(* IEC 61131-3 sources: SmartHomeNew/snapshots/2026-04-28, 18 files *)

(* ---- E_Rule_Comparison.dut ---- *)
{attribute 'strict'}
TYPE E_Rule_Comparison :
(
    COMP_NONE := 0,
    COMP_EQ := 1,
    COMP_GT := 2,
    COMP_LT := 3,
    COMP_GE := 4,
    COMP_LE := 5,
    COMP_IN_RANGE := 6,
    COMP_TRUE := 7,
    COMP_FALSE := 8
) USINT;
END_TYPE

(* ---- E_SENSOR_TYPE.dut ---- *)
{attribute 'strict'}
TYPE E_SENSOR_TYPE :
(
  SENSOR_TYPE_NONE := 0,
  SENSOR_TYPE_DOOR_WINDOW := 5,
  SENSOR_TYPE_GLASS_BREAK := 6,
  SENSOR_TYPE_FLOOD := 7,
  SENSOR_TYPE_SMOKE := 8,
  SENSOR_TYPE_GAS_METHANE := 1,
  SENSOR_TYPE_GAS_CO := 2,
  SENSOR_TYPE_TEMP_FLOOR := 3,
  SENSOR_TYPE_TEMP_AIR := 4,
  SENSOR_TYPE_CO2 := 9
) USINT;
END_TYPE

(* ---- ST_Calibration_Family_Summary.dut ---- *)
{attribute 'pack_mode' := '1'}
TYPE ST_Calibration_Family_Summary :
STRUCT
    active : BOOL;
    status : INT; // 0=OK,1=IN_PROGRESS,2=WARNING,3=ERROR
    sensor_count : INT;
    verification_active_count : INT;
    failed_count : INT;
    max_deviation_percent : REAL;
    summary_text : STRING(160);
END_STRUCT
END_TYPE

(* ---- ST_Gas_Valve_Configuration.dut ---- *)
{attribute 'pack_mode' := '1'}
TYPE ST_Gas_Valve_Configuration :
STRUCT
    valve_id : BYTE := 0;
    valve_type : E_VALVE_TYPE := E_VALVE_TYPE.VALVE_NC;
    close_time_seconds : UDINT := 10;
    open_time_seconds : UDINT := 10;
    emergency_open_allowed : BOOL := FALSE;
END_STRUCT
END_TYPE

(* ---- GVL_HEATING_POLICY.gvl ---- *)
{attribute 'qualified_only'}
VAR_GLOBAL
    G_Zone_Empty_Duration_MS : ARRAY[1..GVL_CONSTANTS.C_MAX_ZONES] OF UDINT;
    G_Zone_Permanent_Use : ARRAY[1..GVL_CONSTANTS.C_MAX_ZONES] OF BOOL;
    G_Zone_Guest_Preheat_Request : ARRAY[1..GVL_CONSTANTS.C_MAX_ZONES] OF BOOL;
    G_Zone_Policy_Class : ARRAY[1..GVL_CONSTANTS.C_MAX_ZONES] OF INT;
    G_Zone_Target_Adjustment : ARRAY[1..GVL_CONSTANTS.C_MAX_ZONES] OF REAL;
    G_Zone_Priority_Bias : ARRAY[1..GVL_CONSTANTS.C_MAX_ZONES] OF REAL;
END_VAR

(* ---- GVL_HEATING_POLICY_CONFIG.gvl ---- *)
{attribute 'qualified_only'}
VAR_GLOBAL
    G_Guest_Preheat_Enabled : BOOL := TRUE;
    G_Guest_Preheat_Priority_Boost : INT := 2;
    G_Guest_Preheat_Max_Duration_MS : UDINT := 7200000; // 2 hours (future use)
END_VAR

(* ---- GVL_INTENT_USER.gvl ---- *)
VAR_GLOBAL
    I_Source_Valid : BOOL := FALSE;
    I_Last_Update_Cycle : UDINT := 0;
    I_Last_Update_MS : UDINT := 0;

    I_Arm_Request : BOOL := FALSE;
    I_Disarm_Request : BOOL := FALSE;

    I_PIN_Code : STRING(8);
    I_RFID_Tag : STRING(32);
    I_2FA_Code_In : STRING(8);

    I_Gate_Open_Request : BOOL := FALSE;
    I_Wicket_Open_Request : BOOL := FALSE;

    I_Lock_1_Open_Request : BOOL := FALSE;
    I_Lock_1_Close_Request : BOOL := FALSE;
    I_Lock_2_Open_Request : BOOL := FALSE;
    I_Lock_2_Close_Request : BOOL := FALSE;

    I_Dangerous_Action_Request : BOOL := FALSE;
    I_Dangerous_Action_Confirm : BOOL := FALSE;
    I_User_Access_Level : INT := 0;

    I_Water_Valve_Test_Open : BOOL := FALSE;
    I_Water_Valve_Test_Close : BOOL := FALSE;
    I_Water_Valve_Test_Confirm : BOOL := FALSE;

    I_Gas_Valve_Test_Open : BOOL := FALSE;
    I_Gas_Valve_Test_Close : BOOL := FALSE;
    I_Gas_Valve_Test_Confirm : BOOL := FALSE;

    I_Water_Selective_Recover : BOOL := FALSE;
    I_Gas_Selective_Recover : BOOL := FALSE;
    I_Scenario_Request : E_SCENARIO_TYPE := E_SCENARIO_TYPE.SCENARIO_NONE;
    I_Lighting_Override_32 : ARRAY[1..32] OF BYTE;
    I_Blinds_Override_32 : ARRAY[1..GVL_CONSTANTS.C_MAX_BLINDS] OF BYTE;
    I_Socket_Override_32 : ARRAY[1..GVL_CONSTANTS.C_MAX_SOCKETS] OF BOOL;
    I_Reset_Errors : BOOL := FALSE;

    I_Set_Temp_Req : BOOL := FALSE;
    I_Target_Zone : INT := 0;
    I_Target_Temperature : REAL := 0.0;
    I_Set_Vent_Req : BOOL := FALSE;
    I_Target_Vent_Speed : REAL := 0.0;
    I_Set_Config_Req : BOOL := FALSE;
    I_Time_Sync_Req : BOOL := FALSE;
    I_New_Time_MS : UDINT := 0;
END_VAR

(* ---- GVL_TEST_PANEL_DEBUG.gvl ---- *)
{attribute 'qualified_only'}
VAR_GLOBAL
    // === DEBUG VIEW ONLY ===
    G_Test_Description : STRING(200);
    G_Test_What_To_Change : STRING(200);
    G_Test_Expected_Text : STRING(200);
    G_Expected_Summary : STRING(200);
    G_Actual_Summary : STRING(200);
    G_Error_Text : STRING(200);
    G_System_State_Line : STRING(200);

    // Inputs snapshot
    G_Input_Guest_Preheat_Request : BOOL;
    G_Input_Guest_Preheat_Enabled : BOOL;
    G_Input_Guest_Preheat_Boost : INT;
    G_Input_Max_Thermal_Budget : REAL;
    G_Input_Block_Heating : BOOL;
    G_Input_Safety_Stop : BOOL;
END_VAR

(* ---- FB_Heating_System_Manager.st ---- *)
// ==============================================================================
// Блок управления системой отопления (Heating System Manager)
// Назначение:
// - Управление контурами теплого пола (открытие/закрытие клапанов).
// - Управление насосами коллекторов и смесительными узлами.
// - Управление каскадом котлов (ротация, расчет ресурса).
// - Защита от перегрева и замерзания.
// - Интеграция с Rule Engine.
// ==============================================================================
FUNCTION_BLOCK FB_Heating_System_Manager
VAR_INPUT
    VI_Preheat_Request : BOOL; // preheat scenario trigger
    L_Climate_Zone_ID : INT;

    VI_System_Mode : E_System_Operating_Mode; // System mode from State Manager

    VI_System_Time_MS : UDINT; // Системное время (мс)
    VI_Current_TOD : TOD; // Текущее время суток
    VI_IsActivePLC : BOOL; // Флаг: Данный ПЛК является ведущим
    VI_Outdoor_Temp : REAL; // Уличная температура воздуха (°C)
    VI_Config : ST_Heating_Config; // Конфигурация системы отопления
    VI_Tariff : ST_Tariff_Config; // Настройки тарифов
    VI_Current_Hour : UINT; // Текущий час (0-23)
    VI_Boiler_Stop : BOOL; // Команда на остановку котлов (от газовой/пожарной сигнализации); вход сохранён для совместимости, не используется как direct control
    VI_DHW_Heating_Demand : BOOL; // Запрос тепла от бойлера ГВС (приоритет)
    VI_DHW_Target_Temp : REAL; // Целевая температура бойлера ГВС
    VI_Current_Scenario : E_SCENARIO_TYPE; // Текущий сценарий
    VI_Emergency_Stop : BOOL; // Агрегированный аварийный стоп от подсистемы безопасности
    VI_Gas_Safety_Stop : BOOL; // Газовая авария / закрытие газового клапана
    VI_Boiler_Error_Status : ARRAY[1..GVL_CONSTANTS.C_MAX_BOILERS] OF BOOL; // Ошибки котлов / ошибка адаптера
    VI_Boiler_OT_Online : ARRAY[1..GVL_CONSTANTS.C_MAX_BOILERS] OF BOOL; // Признак доступности OpenTherm-канала
    VI_Boiler_Modulation : ARRAY[1..GVL_CONSTANTS.C_MAX_BOILERS] OF REAL; // Текущая модуляция котлов (%)
END_VAR
VAR_IN_OUT
    VI_Floor_Temps : ARRAY[1..GVL_CONSTANTS.C_MAX_HEATING_CIRCUITS] OF REAL; // Температуры стяжки пола по зонам
    VI_Room_Temps : ARRAY[1..16] OF REAL; // Температуры воздуха в помещениях
    VI_Manifold_Pressures : ARRAY[1..GVL_CONSTANTS.C_MAX_MANIFOLDS] OF REAL; // Давление в коллекторах (бар)
    VI_Manifold_Currents : ARRAY[1..GVL_CONSTANTS.C_MAX_MANIFOLDS] OF REAL; // Ток насосов коллекторов (мА)
    VI_Manifold_Temps_Supply : ARRAY[1..GVL_CONSTANTS.C_MAX_MANIFOLDS] OF REAL; // Температура подачи на коллекторах
    VI_Manifold_Temps_Return : ARRAY[1..GVL_CONSTANTS.C_MAX_MANIFOLDS] OF REAL; // Температура обратки на коллекторах
    VI_Boiler_Flame_Status : ARRAY[1..GVL_CONSTANTS.C_MAX_BOILERS] OF BOOL; // Статус наличия пламени в котлах
    VI_Zone_Configs : ARRAY[1..GVL_CONSTANTS.C_MAX_HEATING_CIRCUITS] OF ST_FloorHeating_Circuit_Config; // Конфигурации контуров
    VI_Rule_Actions : ARRAY[1..GVL_CONSTANTS.C_MAX_RULES] OF ST_Rule_Action; // Действия от Rule Engine
    VI_IO_Modules_Online : ARRAY[1..GVL_CONSTANTS.C_MAX_MODULES] OF BOOL; // Статусы модулей ввода-вывода
    VI_Scenario_Configs : ARRAY[1..GVL_CONSTANTS.C_MAX_SCENARIOS] OF ST_Scenario_Config; // Конфигурации сценариев
    VI_Manifold_End_Switches : ARRAY[1..GVL_CONSTANTS.C_MAX_MANIFOLDS] OF BOOL; // Концевики клапанов
    VI_Valve_Test_Config : ARRAY[1..GVL_CONSTANTS.C_MAX_MANIFOLDS] OF ST_Valve_Test_Config; // Конфигурация тестирования клапанов
END_VAR

VAR_OUTPUT
    VO_Manifold_Valves : ARRAY[1..GVL_CONSTANTS.C_MAX_MANIFOLDS] OF REAL; // Выход: Положение клапанов смесителей (0-100%)
    VO_Manifold_Pumps : ARRAY[1..GVL_CONSTANTS.C_MAX_MANIFOLDS] OF BOOL; // Выход: Управление насосами коллекторов
    VO_Zone_Valves : ARRAY[1..GVL_CONSTANTS.C_MAX_HEATING_CIRCUITS] OF BOOL; // Выход: Управление клапанами контуров (Зоны 1-16)
    VO_Boiler_OT_Enable : ARRAY[1..GVL_CONSTANTS.C_MAX_BOILERS] OF BOOL; // Физические команды в OpenTherm
    VO_Boiler_OT_Setpoint : ARRAY[1..GVL_CONSTANTS.C_MAX_BOILERS] OF REAL; // Физические уставки в OpenTherm
    VO_Backup_Circulation_Pump : BOOL; // Резервный циркуляционный насос в режиме антизамерзания при газовой аварии
    VO_Electric_Heater_Enable : BOOL; // Сухой контакт электрического нагревателя антизамерзания
    VO_Freeze_Risk_Status : BOOL; // Признак риска замерзания при защёлкнутой газовой аварии
    VO_Status : ARRAY[1..GVL_CONSTANTS.C_MAX_MANIFOLDS] OF ST_Manifold_Status; // Сводный статус коллекторных узлов для HMI
    VO_Boiler_Status : ARRAY[1..GVL_CONSTANTS.C_MAX_BOILERS] OF ST_Boiler_Status; // Сводный статус котлов для HMI
END_VAR

VAR

    L_PID_Valves : ARRAY[1..GVL_CONSTANTS.C_MAX_MANIFOLDS] OF FB_PID_Controller; // ПИД-регуляторы для поддержания температуры подачи
    L_PID_Timer : ARRAY[1..GVL_CONSTANTS.C_MAX_MANIFOLDS] OF FB_System_Timer; // Таймеры вызова ПИД-регуляторов
    L_Floor_Controllers : ARRAY[1..GVL_CONSTANTS.C_MAX_HEATING_CIRCUITS] OF FB_FloorHeating_Controller; // Контроллеры зон теплого пола
    L_Last_Boiler_Rotation : UDINT; // Время последней ротации ведущего котла
    L_Lead_Boiler : BYTE := 1; // Номер ведущего котла (1 или 2)
    L_i : INT; // Индекс для циклов
    L_Zone_Config : ST_FloorHeating_Circuit_Config;
    L_j : INT; // Вспомогательный индекс
    L_Target_Supply_Temp : REAL; // Рассчитанная целевая температура подачи
    L_Demand_Power : REAL; // Суммарный запрос мощности от всех коллекторов
    L_Any_Zone_Active : ARRAY[1..GVL_CONSTANTS.C_MAX_MANIFOLDS] OF BOOL; // Флаги наличия запроса тепла по коллекторам
    L_Current_Temp : REAL; // Текущая температура для ПИД
    L_Sensor_Error : BOOL; // Ошибка обоих датчиков

    // Плавный переход сценария
    L_Prev_Scenario : E_SCENARIO_TYPE;
    L_Scenario_Adjust : REAL;
    L_Target_Scenario_Adjust : REAL;
    L_Transition_Temp : FB_Scenario_Transition_Controller;

    // ТЗ 2.5: Защита от перегрева стяжки
    L_Overheat_Timer : ARRAY[1..GVL_CONSTANTS.C_MAX_HEATING_CIRCUITS] OF FB_System_Timer; // Таймеры задержки отключения при перегреве

    // ТЗ 2.6: Сервисная диагностика и паузы
    L_Pump_Run_Timer : ARRAY[1..GVL_CONSTANTS.C_MAX_MANIFOLDS] OF FB_System_Timer; // Таймер непрерывной работы насоса (до 72ч)
    L_Pump_Pause_Timer : ARRAY[1..GVL_CONSTANTS.C_MAX_MANIFOLDS] OF FB_System_Timer; // Таймер обязательной паузы насоса (1ч)
    L_Pump_In_Pause : ARRAY[1..GVL_CONSTANTS.C_MAX_MANIFOLDS] OF BOOL; // Флаг: Насос находится в режиме сервисной паузы

    // ТЗ 2.8: Учет ресурса оборудования
    L_Last_Scan_Time : UDINT; // Время предыдущего цикла для расчета наработки
    L_Scan_Time_Init : BOOL := FALSE;
    L_Lifespan_S : REAL := 50000.0 * 3600.0; // Расчетный ресурс котла (50,000 часов в секундах)
    L_Delta_MS : UDINT; // Разница времени
    L_Pump_Diag : ARRAY[1..GVL_CONSTANTS.C_MAX_MANIFOLDS] OF FB_Device_Predictive_Diag; // Диагностика насосов
    L_Boiler_Life : ARRAY[1..GVL_CONSTANTS.C_MAX_BOILERS] OF FB_Lifetime_Predictor; // Предиктор ресурса котлов

    fbFloorTempValidator : ARRAY[1..GVL_CONSTANTS.C_MAX_HEATING_CIRCUITS] OF FB_Analog_Validator;
    fbRoomTempValidator : ARRAY[1..16] OF FB_Analog_Validator;
    fbValveTestManager : FB_Valve_Test_Manager; // Менеджер тестирования клапанов
    fbBoilerCascade : FB_Boiler_Cascade_Manager; // Выделенный менеджер каскада котлов
    fbBoilerOpenTherm : FB_Boiler_OpenTherm_Interface; // Основной транспорт OpenTherm
    L_IO_Failsafe_Active : BOOL; // Флаг потери связи с модулями I/O
    L_Freeze_Mode_Active : BOOL; // Флаг антизамерзания по ТЗ
    L_Freeze_Target_Supply : REAL; // Уставка подачи в режиме антизамерзания
    L_Delta_T : REAL; // Разница температур подача/обратка
    L_Min_Supply_Temp : REAL; // Минимальная температура теплоносителя для антизамерзания
    L_Boiler_OT_Command_Valid : ARRAY[1..GVL_CONSTANTS.C_MAX_BOILERS] OF BOOL; // Команда ушла через OT
    L_Boiler_Request_Enable : ARRAY[1..GVL_CONSTANTS.C_MAX_BOILERS] OF BOOL; // Внутренний request на котлы от логики каскада
    L_Boiler_Request_Setpoint : ARRAY[1..GVL_CONSTANTS.C_MAX_BOILERS] OF REAL; // Внутренняя request-уставка котлов
    L_Policy_Normal : BOOL; // Policy: normal operation
    L_Policy_Safe_Stop : BOOL; // Policy: hard safe stop
    L_Policy_Degraded : BOOL; // Policy: limited conservative operation
    L_Policy_Freeze_Protection : BOOL; // Policy: freeze protection mode
    L_Any_Sensor_Error : BOOL;
    L_Any_Subsystem_Degraded : BOOL;
    L_Adaptive_Max_Delta : REAL;
    L_Adaptive_Delta : REAL;
    L_Adaptive_Zone_i : INT;
    L_Adaptive_Weighted_Sum : REAL;
    L_Adaptive_Weight_Total : REAL;
    L_Adaptive_Effective_Delta : REAL;
    L_Adaptive_Weight : REAL;
    L_Adaptive_Correction : REAL;
END_VAR

// ========================================
// Heating policy layer
// ========================================
L_Policy_Normal := (VI_System_Mode = E_System_Operating_Mode.MODE_NORMAL);
L_Policy_Safe_Stop := (VI_System_Mode = E_System_Operating_Mode.MODE_SAFE_STOP);
L_Policy_Degraded := (VI_System_Mode = E_System_Operating_Mode.MODE_DEGRADED);
L_Policy_Freeze_Protection := (VI_System_Mode = E_System_Operating_Mode.MODE_FREEZE_PROTECTION);

// ========================================
// Heating freeze policy activation
// ========================================
IF L_Policy_Freeze_Protection THEN
    L_Freeze_Mode_Active := TRUE;
END_IF;

// 0. Агрегация деградации для system mode
GVL_STATE.G_Heating_IO_Fault := FALSE;
GVL_STATE.G_Heating_Sensor_Fault := FALSE;
GVL_STATE.G_Heating_Subsystem_Degraded := FALSE;
L_Any_Sensor_Error := FALSE;
L_Any_Subsystem_Degraded := FALSE;

// 0. Аварийный стоп от подсистемы безопасности
VO_Backup_Circulation_Pump := FALSE;
VO_Electric_Heater_Enable := FALSE;
VO_Freeze_Risk_Status := FALSE;

IF VI_Gas_Safety_Stop THEN
    L_Freeze_Mode_Active := (VI_Outdoor_Temp < -5.0);
    FOR L_i := 1 TO GVL_CONSTANTS.C_MAX_HEATING_CIRCUITS DO
        IF VI_Floor_Temps[L_i] < 7.0 THEN
            L_Freeze_Mode_Active := TRUE;
        END_IF;
        VO_Zone_Valves[L_i] := FALSE;
    END_FOR;

    FOR L_i := 1 TO GVL_CONSTANTS.C_MAX_MANIFOLDS DO
        VO_Manifold_Pumps[L_i] := FALSE;
        VO_Manifold_Valves[L_i] := 0.0;
    END_FOR;

    FOR L_i := 1 TO GVL_CONSTANTS.C_MAX_BOILERS DO
        VO_Boiler_OT_Enable[L_i] := FALSE;
        VO_Boiler_OT_Setpoint[L_i] := 0.0;
        VO_Boiler_Status[L_i].Warning := FALSE;
        VO_Boiler_Status[L_i].Error := TRUE;
    END_FOR;

    IF L_Freeze_Mode_Active THEN
        VO_Backup_Circulation_Pump := TRUE;
        L_Freeze_Target_Supply := LIMIT(20.0, VI_Config.Freeze_Threshold + 2.0, 35.0);
        L_Min_Supply_Temp := 1000.0;
        FOR L_i := 1 TO GVL_CONSTANTS.C_MAX_MANIFOLDS DO
            IF VI_Manifold_Temps_Supply[L_i] < L_Min_Supply_Temp THEN
                L_Min_Supply_Temp := VI_Manifold_Temps_Supply[L_i];
            END_IF;
        END_FOR;
        IF L_Min_Supply_Temp > 900.0 THEN
            L_Min_Supply_Temp := 0.0;
        END_IF;

        IF L_Min_Supply_Temp < (L_Freeze_Target_Supply - 1.0) THEN
            VO_Electric_Heater_Enable := TRUE;
        ELSIF L_Min_Supply_Temp > (L_Freeze_Target_Supply + 1.0) THEN
            VO_Electric_Heater_Enable := FALSE;
        END_IF;

        // При защёлкнутой газовой аварии оператор должен видеть, что система живёт в деградированном anti-freeze режиме.
        VO_Freeze_Risk_Status := TRUE;
    END_IF;

    RETURN;
END_IF;

IF VI_Emergency_Stop OR L_Policy_Safe_Stop THEN
    FOR L_i := 1 TO GVL_CONSTANTS.C_MAX_HEATING_CIRCUITS DO
        VO_Zone_Valves[L_i] := FALSE;
    END_FOR;

    FOR L_i := 1 TO GVL_CONSTANTS.C_MAX_MANIFOLDS DO
        VO_Manifold_Pumps[L_i] := FALSE;
        VO_Manifold_Valves[L_i] := 0.0;
    END_FOR;

    FOR L_i := 1 TO GVL_CONSTANTS.C_MAX_BOILERS DO
        VO_Boiler_OT_Enable[L_i] := FALSE;
        VO_Boiler_OT_Setpoint[L_i] := 0.0;
        VO_Boiler_Status[L_i].Warning := FALSE;
        VO_Boiler_Status[L_i].Error := TRUE;
    END_FOR;

    RETURN;
END_IF;

// 1. Проверка связи с модулями ввода-вывода (ТЗ 2.0)
L_IO_Failsafe_Active := FALSE;
FOR L_i := 1 TO GVL_CONSTANTS.C_MAX_MODULES DO
    IF NOT VI_IO_Modules_Online[L_i] THEN
        L_IO_Failsafe_Active := TRUE;
        GVL_STATE.G_Heating_IO_Fault := TRUE;
GVL_STATE.G_Heating_Subsystem_Degraded := TRUE;
        EXIT;
    END_IF;
END_FOR;

IF L_IO_Failsafe_Active THEN
    // Fail-safe: закрываем зональные клапаны, чтобы не разгонять неконтролируемые контуры,
    // но при риске замерзания сохраняем минимальную циркуляцию и минимальную теплогенерацию.
    L_Freeze_Mode_Active := (VI_Outdoor_Temp < -5.0);

    FOR L_j := 1 TO GVL_CONSTANTS.C_MAX_HEATING_CIRCUITS DO
        IF VI_Floor_Temps[L_j] < 7.0 THEN
            L_Freeze_Mode_Active := TRUE;
        END_IF;
        VO_Zone_Valves[L_j] := FALSE;
    END_FOR;

    IF L_Freeze_Mode_Active THEN
        L_Freeze_Target_Supply := LIMIT(20.0, VI_Config.Freeze_Threshold + 2.0, 35.0);
    ELSE
        L_Freeze_Target_Supply := 0.0;
    END_IF;

    FOR L_j := 1 TO GVL_CONSTANTS.C_MAX_MANIFOLDS DO
        IF L_Freeze_Mode_Active THEN
            VO_Manifold_Pumps[L_j] := TRUE;
            VO_Manifold_Valves[L_j] := 35.0;
        ELSE
            VO_Manifold_Pumps[L_j] := FALSE;
            VO_Manifold_Valves[L_j] := 0.0;
        END_IF;
    END_FOR;

    // В аварийном I/O режиме напрямую формируем только legacy request-мirror.
    // Реальные физические команды всё равно будут интерпретированы transport-слоем выше по архитектуре.
    FOR L_j := 1 TO GVL_CONSTANTS.C_MAX_BOILERS DO
        VO_Boiler_OT_Enable[L_j] := FALSE;
        VO_Boiler_OT_Setpoint[L_j] := 0.0;
    END_FOR;

    IF L_Freeze_Mode_Active THEN
        // В fail-safe используем только ведущий аварийный вариант: котёл №1 на минимальной уставке.
        IF VI_Boiler_OT_Online[1] AND NOT VI_Boiler_Error_Status[1] THEN
            VO_Boiler_OT_Enable[1] := TRUE;
            VO_Boiler_OT_Setpoint[1] := L_Freeze_Target_Supply;
        END_IF;
    END_IF;

    RETURN;
END_IF;

// --- HEATING TARGET INJECTION ---
// Global arbitration target is applied after base policy calculation.
IF GVL_STATE.G_Target_Temperature > 0.0 THEN
    L_Target_Supply_Temp := GVL_STATE.G_Target_Temperature;
END_IF;

// --- MULTI-ZONE ADAPTIVE CORRECTION ---
// Final adaptive refinement layer.
L_Adaptive_Max_Delta := 0.0;
L_Adaptive_Weighted_Sum := 0.0;
L_Adaptive_Weight_Total := 0.0;
L_Adaptive_Effective_Delta := 0.0;
L_Adaptive_Correction := 0.0;

FOR L_Adaptive_Zone_i := 1 TO GVL_CONSTANTS.C_MAX_HEATING_CIRCUITS DO
    IF VI_Zone_Configs[L_Adaptive_Zone_i].zone >= 1 AND VI_Zone_Configs[L_Adaptive_Zone_i].zone <= 8 THEN
        CASE VI_Zone_Configs[L_Adaptive_Zone_i].control_type OF
            0:
                L_Adaptive_Delta :=
                    VI_Zone_Configs[L_Adaptive_Zone_i].design_temp -
                    VI_Floor_Temps[L_Adaptive_Zone_i];
                L_Adaptive_Weight := 0.6;
            1, 2:
                L_Adaptive_Delta :=
                    VI_Zone_Configs[L_Adaptive_Zone_i].design_temp -
                    VI_Room_Temps[VI_Zone_Configs[L_Adaptive_Zone_i].zone];
                L_Adaptive_Weight := 1.0;
            ELSE
                L_Adaptive_Delta :=
                    VI_Zone_Configs[L_Adaptive_Zone_i].design_temp -
                    VI_Room_Temps[VI_Zone_Configs[L_Adaptive_Zone_i].zone];
                L_Adaptive_Weight := 0.8;
        END_CASE;

        IF VI_Zone_Configs[L_Adaptive_Zone_i].zone >= 1 AND VI_Zone_Configs[L_Adaptive_Zone_i].zone <= 4 THEN
            L_Adaptive_Weight := L_Adaptive_Weight * 1.2;
        ELSIF VI_Zone_Configs[L_Adaptive_Zone_i].zone >= 9 THEN
            L_Adaptive_Weight := L_Adaptive_Weight * 0.7;
        END_IF;

        IF L_Adaptive_Weight > 2.0 THEN
            L_Adaptive_Weight := 2.0;
        ELSIF L_Adaptive_Weight < 0.2 THEN
            L_Adaptive_Weight := 0.2;
        END_IF;

        IF L_Adaptive_Delta > L_Adaptive_Max_Delta THEN
            L_Adaptive_Max_Delta := L_Adaptive_Delta;
        END_IF;

        L_Adaptive_Weighted_Sum := L_Adaptive_Weighted_Sum + (L_Adaptive_Delta * L_Adaptive_Weight);
        L_Adaptive_Weight_Total := L_Adaptive_Weight_Total + L_Adaptive_Weight;
    END_IF;
END_FOR;

IF L_Adaptive_Weight_Total > 0.0 THEN
    L_Adaptive_Effective_Delta := L_Adaptive_Weighted_Sum / L_Adaptive_Weight_Total;
END_IF;

IF L_Adaptive_Effective_Delta > 1.5 THEN
    L_Adaptive_Correction := 2.0;
ELSIF L_Adaptive_Effective_Delta > 0.7 THEN
    L_Adaptive_Correction := 1.0;
ELSIF L_Adaptive_Effective_Delta < -1.5 THEN
    L_Adaptive_Correction := -2.0;
ELSIF L_Adaptive_Effective_Delta < -0.7 THEN
    L_Adaptive_Correction := -1.0;
ELSE
    L_Adaptive_Correction := 0.0;
END_IF;

IF L_Adaptive_Max_Delta > 2.5 AND L_Adaptive_Correction < 2.0 THEN
    L_Adaptive_Correction := 2.0;
END_IF;

L_Target_Supply_Temp := L_Target_Supply_Temp + L_Adaptive_Correction;

IF L_Target_Supply_Temp < 20.0 THEN
    L_Target_Supply_Temp := 20.0;
ELSIF L_Target_Supply_Temp > 45.0 THEN
    L_Target_Supply_Temp := 45.0;
END_IF;

// 2. Индивидуальное управление зонами отопления (ТЗ 1.1, 2.5)
FOR L_i := 1 TO GVL_CONSTANTS.C_MAX_HEATING_CIRCUITS DO
    fbFloorTempValidator[L_i](
        VI_Value := VI_Floor_Temps[L_i],
        VI_Min_Valid := -40.0,
        VI_Max_Valid := 120.0,
        VI_Fallback_Mode := 0
    );

    L_Climate_Zone_ID := VI_Zone_Configs[L_i].zone;
    IF L_Climate_Zone_ID >= 1 AND L_Climate_Zone_ID <= 16 THEN
        fbRoomTempValidator[L_Climate_Zone_ID](
        VI_Value := VI_Room_Temps[L_Climate_Zone_ID],
        VI_Min_Valid := -40.0,
        VI_Max_Valid := 120.0,
        VI_Fallback_Mode := 0
        );
    END_IF;

    // Контроль перегрева стяжки (защита напольного покрытия)
    L_Overheat_Timer[L_i](IN := fbFloorTempValidator[L_i].VO_Value > VI_Config.Overheat_Threshold, PT := T#60s, VI_System_Time_MS := VI_System_Time_MS);

    // Выбор датчика температуры с автоматическим переключением при неисправности
    L_Current_Temp := 0.0;
    L_Sensor_Error := FALSE;

    IF VI_Zone_Configs[L_i].control_type = 1 OR VI_Zone_Configs[L_i].control_type = 2 THEN
        // Основной: по воздуху
        IF NOT fbRoomTempValidator[L_Climate_Zone_ID].VO_Error THEN
            L_Current_Temp := fbRoomTempValidator[L_Climate_Zone_ID].VO_Value;
        ELSIF NOT fbFloorTempValidator[L_i].VO_Error THEN
            L_Current_Temp := fbFloorTempValidator[L_i].VO_Value; // Резервный: по полу
        ELSE
            L_Sensor_Error := TRUE;
        END_IF;
    ELSE
        // Основной: по полу
        IF NOT fbFloorTempValidator[L_i].VO_Error THEN
            L_Current_Temp := fbFloorTempValidator[L_i].VO_Value;
        ELSIF NOT fbRoomTempValidator[L_Climate_Zone_ID].VO_Error THEN
            L_Current_Temp := fbRoomTempValidator[L_Climate_Zone_ID].VO_Value; // Резервный: по воздуху
        ELSE
            L_Sensor_Error := TRUE;
        END_IF;
    END_IF;

    IF L_Sensor_Error THEN
        L_Any_Sensor_Error := TRUE;
        VO_Zone_Valves[L_i] := FALSE; // Безопасное состояние при ошибке обоих датчиков
    ELSE
        // ПИД-регулирование и ШИМ для каждой зоны
        // Применяем плавную корректировку уставки от сценария
        L_Zone_Config := VI_Zone_Configs[L_i];
        L_Zone_Config.design_temp := L_Zone_Config.design_temp + L_Scenario_Adjust;
        L_Floor_Controllers[L_i](
            VI_Current_Temp := L_Current_Temp,
            VI_Config := L_Zone_Config,
            VI_Tariff := VI_Tariff,
            VI_Current_Hour := VI_Current_Hour,
            VI_IsActivePLC := VI_IsActivePLC,
            VI_System_Time_MS := VI_System_Time_MS,
            VO_Valve_Bool => VO_Zone_Valves[L_i]
        );
    END_IF;

    // Принудительное закрытие клапана при перегреве пола (ТЗ 2.5)
    IF L_Overheat_Timer[L_i].Q THEN
        VO_Zone_Valves[L_i] := FALSE;
    END_IF;

    // Обработка действий от Rule Engine (ТЗ 13.0)
    FOR L_j := 1 TO GVL_CONSTANTS.C_MAX_RULES DO
        IF VI_Rule_Actions[L_j].Active AND VI_Rule_Actions[L_j].Target_ID = L_i THEN
            IF VI_Rule_Actions[L_j].Action_Type = E_Rule_Action_Type.ACTION_SET_FLOOR_HEATING THEN
                VO_Zone_Valves[L_i] := (VI_Rule_Actions[L_j].Value > 0.5);
            END_IF;
        END_IF;
    END_FOR;
END_FOR;

GVL_STATE.G_Heating_Sensor_Fault := L_Any_Sensor_Error;

// 3. Определение потребности в работе коллекторных насосов
FOR L_i := 1 TO GVL_CONSTANTS.C_MAX_MANIFOLDS DO
    L_Any_Zone_Active[L_i] := FALSE;
END_FOR;

FOR L_i := 1 TO GVL_CONSTANTS.C_MAX_HEATING_CIRCUITS DO
    IF VO_Zone_Valves[L_i] THEN
        L_j := VI_Zone_Configs[L_i].manifold_id;
        IF L_j >= 1 AND L_j <= GVL_CONSTANTS.C_MAX_MANIFOLDS THEN
            L_Any_Zone_Active[L_j] := TRUE;
        END_IF;
    END_IF;
END_FOR;

// 4. Управление смесительными узлами коллекторов (ТЗ 2.6, 12.2)
FOR L_i := 1 TO GVL_CONSTANTS.C_MAX_MANIFOLDS DO
    // ПИД-регулирование трехходового клапана для поддержания стабильной температуры подачи
    // Вызываем ПИД регулятор каждую секунду
    L_PID_Timer[L_i](IN := TRUE, PT := T#1s, VI_System_Time_MS := VI_System_Time_MS);
    IF L_PID_Timer[L_i].Q THEN
        L_PID_Timer[L_i](IN := FALSE, PT := T#1s, VI_System_Time_MS := VI_System_Time_MS); // Сброс таймера
        L_PID_Timer[L_i](IN := TRUE, PT := T#1s, VI_System_Time_MS := VI_System_Time_MS); // Перезапуск

        L_PID_Valves[L_i](
            VI_SetPoint := L_Target_Supply_Temp,
            VI_ProcessValue := VI_Manifold_Temps_Supply[L_i],
            VI_Kp := 2.0, VI_Tn := 120.0, VI_Tv := 0.0,
            VI_Y_Min := 0.0, VI_Y_Max := 100.0, VI_Cycle_Time_S := 1.0,
            VO_Output => VO_Manifold_Valves[L_i]
        );
    END_IF;

    // ТЗ 2.6: Реализация обязательной паузы насоса (защита от закисания и перегрева при 72ч работе)
    L_Pump_Run_Timer[L_i](IN := VO_Manifold_Pumps[L_i] AND NOT L_Pump_In_Pause[L_i], PT := T#72h, VI_System_Time_MS := VI_System_Time_MS);
    IF L_Pump_Run_Timer[L_i].Q THEN L_Pump_In_Pause[L_i] := TRUE; END_IF;

    L_Pump_Pause_Timer[L_i](IN := L_Pump_In_Pause[L_i], PT := T#1h, VI_System_Time_MS := VI_System_Time_MS);
    IF L_Pump_Pause_Timer[L_i].Q THEN L_Pump_In_Pause[L_i] := FALSE; END_IF;

    // Включение насоса при наличии запроса от зон и отсутствии сервисной паузы
    // Приоритет ГВС: если есть запрос от ГВС, отключаем насосы отопления и закрываем клапаны
    IF VI_DHW_Heating_Demand THEN
        VO_Manifold_Pumps[L_i] := FALSE;
        VO_Manifold_Valves[L_i] := 0.0; // Принудительно закрываем смесительный клапан
    ELSE
        VO_Manifold_Pumps[L_i] := VI_IsActivePLC AND L_Any_Zone_Active[L_i] AND NOT L_Pump_In_Pause[L_i];
    END_IF;

    // Защита от замерзания системы (ТЗ 2.4)
        IF L_Freeze_Mode_Active THEN
            VO_Manifold_Pumps[L_i] := TRUE;
            IF VO_Manifold_Valves[L_i] < 35.0 THEN
                VO_Manifold_Valves[L_i] := 35.0;
            END_IF;
        END_IF;

        // Сбор диагностических данных для визуализации на HMI
    VO_Status[L_i].Pump_On := VO_Manifold_Pumps[L_i];
    VO_Status[L_i].Pump_Current := VI_Manifold_Currents[L_i];
    VO_Status[L_i].Pressure := VI_Manifold_Pressures[L_i];
    VO_Status[L_i].Temp_Supply := VI_Manifold_Temps_Supply[L_i];
    VO_Status[L_i].Temp_Return := VI_Manifold_Temps_Return[L_i];
    VO_Status[L_i].Valve_Pos := VO_Manifold_Valves[L_i];

    // Предиктивная диагностика насоса
    L_Pump_Diag[L_i](
        VI_Current_Value := VI_Manifold_Currents[L_i],
        VI_Nominal_Value := 0.55, // Номинальный ток насоса по ТЗ: середина диапазона 0.3..0.8 А
        VI_Is_Running := VO_Manifold_Pumps[L_i],
        VI_Reset_Stats := FALSE,
        VI_System_Time_MS := VI_System_Time_MS,
        VIO_Health_Data := VO_Status[L_i].Health
    );

    // Автоматический контроль рабочих параметров (ток / давление / ΔT)
        IF VO_Manifold_Pumps[L_i] THEN
            L_Delta_T := VI_Manifold_Temps_Supply[L_i] - VI_Manifold_Temps_Return[L_i];

            // Контроль тока насоса:
            // Приоритет ошибок:
            // 1. Насос/ток
            // 2. Давление
            // 3. ΔT
            VO_Status[L_i].Error := FALSE;
            VO_Status[L_i].Error_ID := 0;

            IF VI_Manifold_Currents[L_i] <= 0.01 THEN
                VO_Status[L_i].Error := TRUE;
                VO_Status[L_i].Error_ID := TO_WORD(GVL_CONFIG.ERR_PUMP_NO_CURRENT);
            ELSIF VI_Manifold_Currents[L_i] < 0.3 THEN
                VO_Status[L_i].Error := TRUE;
                VO_Status[L_i].Error_ID := TO_WORD(GVL_CONFIG.ERR_PUMP_UNDERCURRENT);
            ELSIF VI_Manifold_Currents[L_i] > 1.5 THEN
                VO_Status[L_i].Error := TRUE;
                VO_Status[L_i].Error_ID := TO_WORD(GVL_CONFIG.ERR_PUMP_OVERCURRENT);
            END_IF;

            // Проверка давления в системе (норма 1.5 - 2.5 бар)
            IF (NOT VO_Status[L_i].Error) AND (VI_Manifold_Pressures[L_i] < 1.5 OR VI_Manifold_Pressures[L_i] > 2.5) THEN
                VO_Status[L_i].Error := TRUE;
                VO_Status[L_i].Error_ID := TO_WORD(GVL_CONFIG.ERR_PRESSURE_OUT_OF_RANGE);
            END_IF;

            // Проверка эффективности теплообмена (ΔT 5..10°C норма)
            IF NOT VO_Status[L_i].Error THEN
                IF L_Delta_T < 5.0 THEN
                    VO_Status[L_i].Error := TRUE;
                    VO_Status[L_i].Error_ID := TO_WORD(GVL_CONFIG.ERR_DELTA_T_LOW);
                ELSIF L_Delta_T > 10.0 THEN
                    VO_Status[L_i].Error := TRUE;
                    VO_Status[L_i].Error_ID := TO_WORD(GVL_CONFIG.ERR_DELTA_T_HIGH);
                END_IF;
            END_IF;
        END_IF;

        // ТЗ 12.2: Еженедельное тестирование запорной арматуры (предотвращение закисания)
    // Выполняется менеджером fbValveTestManager
END_FOR;

fbValveTestManager(
    VI_System_Time_MS := VI_System_Time_MS,
    VI_IsActivePLC := VI_IsActivePLC,
    VI_Valve_Currents := VI_Manifold_Currents,
    VI_Valve_End_Switches := VI_Manifold_End_Switches,
    VI_Config := VI_Valve_Test_Config
);

IF fbValveTestManager.VO_Test_Active THEN
    L_i := fbValveTestManager.VO_Current_Valve;
    IF L_i >= 1 AND L_i <= GVL_CONSTANTS.C_MAX_MANIFOLDS THEN
        IF fbValveTestManager.VO_Valve_Cmd[L_i] THEN
            VO_Manifold_Valves[L_i] := 100.0;
        ELSE
            VO_Manifold_Valves[L_i] := 0.0;
        END_IF;
        VO_Manifold_Pumps[L_i] := FALSE; // Отключаем насос при тестировании клапана
    END_IF;
END_IF;

// 5. Управление каскадом котлов (ТЗ 2.8, OpenTherm-only, без legacy mirror)
L_Demand_Power := 0.0;
FOR L_i := 1 TO GVL_CONSTANTS.C_MAX_MANIFOLDS DO
    IF VO_Manifold_Pumps[L_i] THEN
        L_Demand_Power := L_Demand_Power + VO_Manifold_Valves[L_i];
    END_IF;
END_FOR;

// В режиме антизамерзания обеспечиваем минимальный запрос тепла
IF L_Freeze_Mode_Active AND L_Demand_Power < 20.0 THEN
    L_Demand_Power := 20.0;
END_IF;

IF L_Policy_Degraded THEN
    IF L_Demand_Power > 60.0 THEN
        L_Demand_Power := 60.0;
    END_IF;
END_IF;

fbBoilerCascade(
    VI_Enable := VI_IsActivePLC AND ((L_Demand_Power > GVL_CONSTANTS.C_BOILER_CASCADE_MIN_DEMAND) OR L_Freeze_Mode_Active),
    VI_System_Time_MS := VI_System_Time_MS,
    VI_Boiler_Stop := FALSE,
    VI_DHW_Heating_Demand := VI_DHW_Heating_Demand,
    VI_DHW_Target_Temp := VI_DHW_Target_Temp,
    VI_Target_Supply_Temp := L_Target_Supply_Temp,
    VI_Demand_Power := L_Demand_Power,
    VI_Boiler_Flame_Status := VI_Boiler_Flame_Status,
    VI_Boiler_Error_Status := VI_Boiler_Error_Status,
    VI_Boiler_OT_Online := VI_Boiler_OT_Online,
    VI_Boiler_Modulation := VI_Boiler_Modulation,
    VO_Boiler_Enable => L_Boiler_Request_Enable,
    VO_Boiler_Setpoint => L_Boiler_Request_Setpoint,
    VO_Lead_Boiler => L_Lead_Boiler
);

// ========================================
// OT availability enforcement (no fallback)
// ========================================
FOR L_i := 1 TO GVL_CONSTANTS.C_MAX_BOILERS DO
    IF NOT VI_Boiler_OT_Online[L_i] OR VI_Boiler_Error_Status[L_i] THEN
        L_Boiler_Request_Enable[L_i] := FALSE;
        L_Boiler_Request_Setpoint[L_i] := 0.0;
    END_IF;
END_FOR;

fbBoilerOpenTherm(
    VI_Enable := L_Boiler_Request_Enable,
    VI_Setpoint := L_Boiler_Request_Setpoint,
    VI_OT_Online := VI_Boiler_OT_Online,
    VI_OT_Error := VI_Boiler_Error_Status,
    VO_OT_Enable => VO_Boiler_OT_Enable,
    VO_OT_Setpoint => VO_Boiler_OT_Setpoint,
    VO_OT_Command_Valid => L_Boiler_OT_Command_Valid
);

// ========================================
// Boiler status normalization
// ========================================
FOR L_i := 1 TO GVL_CONSTANTS.C_MAX_BOILERS DO
    // Базовый сброс диагностических флагов котла
    VO_Boiler_Status[L_i].Active := L_Boiler_Request_Enable[L_i];
    VO_Boiler_Status[L_i].Warning := FALSE;
    VO_Boiler_Status[L_i].Error := FALSE;

    // Приоритет причин:
    // 1. Нет канала OpenTherm
    // 2. Котёл вернул ошибку
    // 3. Есть запрос, но нет пламени
    IF NOT VI_Boiler_OT_Online[L_i] THEN
        VO_Boiler_Status[L_i].Error := TRUE;
        VO_Boiler_Status[L_i].Error_ID := TO_WORD(GVL_CONFIG.ERR_BOILER_OFFLINE);
        L_Any_Subsystem_Degraded := TRUE;
    ELSIF VI_Boiler_Error_Status[L_i] THEN
        VO_Boiler_Status[L_i].Error := TRUE;
        VO_Boiler_Status[L_i].Error_ID := TO_WORD(GVL_CONFIG.ERR_BOILER_GENERAL_FAULT);
        L_Any_Subsystem_Degraded := TRUE;
    ELSIF L_Boiler_Request_Enable[L_i] AND NOT VI_Boiler_Flame_Status[L_i] THEN
        VO_Boiler_Status[L_i].Warning := TRUE;
        VO_Boiler_Status[L_i].Error_ID := TO_WORD(GVL_CONFIG.ERR_BOILER_NO_FLAME);
        L_Any_Subsystem_Degraded := TRUE;
    ELSE
        VO_Boiler_Status[L_i].Error_ID := 0;
    END_IF;
END_FOR;

// Расчет наработки и остаточного ресурса котлов (ТЗ 2.8)
IF NOT L_Scan_Time_Init THEN
    L_Last_Scan_Time := VI_System_Time_MS;
    L_Scan_Time_Init := TRUE;
END_IF;

L_Delta_MS := (SEL(VI_System_Time_MS >= L_Last_Scan_Time, VI_System_Time_MS - L_Last_Scan_Time, (4294967295 - L_Last_Scan_Time) + VI_System_Time_MS + 1));
IF L_Delta_MS > 1000 THEN
    L_Delta_MS := 1000; // Ограничение дельты для предотвращения скачков после перезагрузки
END_IF;

L_Last_Scan_Time := VI_System_Time_MS;

FOR L_i := 1 TO GVL_CONSTANTS.C_MAX_BOILERS DO
    VO_Boiler_Status[L_i].Work_Seconds := GVL_Retain.G_Boiler_Work_Seconds[L_i];

    IF VI_Boiler_Flame_Status[L_i] THEN
        GVL_Retain.G_Boiler_Accumulated_MS[L_i] := GVL_Retain.G_Boiler_Accumulated_MS[L_i] + L_Delta_MS;
        IF GVL_Retain.G_Boiler_Accumulated_MS[L_i] >= GVL_CONSTANTS.C_MS_IN_SECOND THEN
            GVL_Retain.G_Boiler_Work_Seconds[L_i] := GVL_Retain.G_Boiler_Work_Seconds[L_i] + (GVL_Retain.G_Boiler_Accumulated_MS[L_i] / 1000);
            GVL_Retain.G_Boiler_Accumulated_MS[L_i] := GVL_Retain.G_Boiler_Accumulated_MS[L_i] MOD 1000;

            // Защита от переполнения (сброс при достижении ~136 лет)
            IF GVL_Retain.G_Boiler_Work_Seconds[L_i] > 4000000000 THEN
                GVL_Retain.G_Boiler_Work_Seconds[L_i] := 0;
            END_IF;

            VO_Boiler_Status[L_i].Work_Seconds := GVL_Retain.G_Boiler_Work_Seconds[L_i];
        END_IF;
    END_IF;

    VO_Boiler_Status[L_i].Work_Hours := TO_REAL(VO_Boiler_Status[L_i].Work_Seconds) / 3600.0;

    L_Boiler_Life[L_i](
        VI_Runtime_Hours := TO_UDINT(VO_Boiler_Status[L_i].Work_Hours),
        VI_Start_Count := 0, // Не считаем пуски для котлов в этой версии
        VI_Nominal_Life := 50000 // 50,000 часов
    );
    VO_Boiler_Status[L_i].Resource_Percent := TO_REAL(L_Boiler_Life[L_i].VO_Remaining_Percent);
    VO_Boiler_Status[L_i].Running := VI_Boiler_Flame_Status[L_i];
END_FOR;
GVL_STATE.G_Heating_Subsystem_Degraded := L_Any_Subsystem_Degraded;

END_FUNCTION_BLOCK
// >>> BULK_SYNC_ANCHOR: FB_Heating_System_Manager <<<

(* ---- FB_Safety_Workflow_Manager.st ---- *)
FUNCTION_BLOCK FB_Safety_Workflow_Manager
VAR_INPUT
    VI_System_Time_MS : UDINT;
    VI_Water_Selective_Recover : BOOL;
    VI_Gas_Selective_Recover : BOOL;
    VI_Water_Valve_Test_Open : BOOL;
    VI_Water_Valve_Test_Close : BOOL;
    VI_Water_Valve_Test_Confirm : BOOL;
    VI_Gas_Valve_Test_Open : BOOL;
    VI_Gas_Valve_Test_Close : BOOL;
    VI_Gas_Valve_Test_Confirm : BOOL;
END_VAR
VAR_OUTPUT
    VO_Water_Selective_Recover_Edge : BOOL;
    VO_Gas_Selective_Recover_Edge : BOOL;
    VO_Water_Valve_Test_Open_Edge : BOOL;
    VO_Water_Valve_Test_Close_Edge : BOOL;
    VO_Water_Valve_Test_Confirm_Edge : BOOL;
    VO_Gas_Valve_Test_Open_Edge : BOOL;
    VO_Gas_Valve_Test_Close_Edge : BOOL;
    VO_Gas_Valve_Test_Confirm_Edge : BOOL;
    VO_Water_Test_Active : BOOL;
    VO_Gas_Test_Active : BOOL;
    VO_Water_Test_Timeout_Close_Required : BOOL;
    VO_Gas_Test_Timeout_Close_Required : BOOL;
END_VAR
VAR
    L_CMD_Water_Selective_Recover_Prev : BOOL;
    L_CMD_Gas_Selective_Recover_Prev : BOOL;
    L_CMD_Water_Valve_Test_Open_Prev : BOOL;
    L_CMD_Water_Valve_Test_Close_Prev : BOOL;
    L_CMD_Water_Valve_Test_Confirm_Prev : BOOL;
    L_CMD_Gas_Valve_Test_Open_Prev : BOOL;
    L_CMD_Gas_Valve_Test_Close_Prev : BOOL;
    L_CMD_Gas_Valve_Test_Confirm_Prev : BOOL;
    L_Water_Test_Active : BOOL;
    L_Water_Test_Deadline : UDINT;
    L_Gas_Test_Active : BOOL;
    L_Gas_Test_Deadline : UDINT;
END_VAR

VO_Water_Test_Timeout_Close_Required := FALSE;
VO_Gas_Test_Timeout_Close_Required := FALSE;

VO_Water_Selective_Recover_Edge := VI_Water_Selective_Recover AND NOT L_CMD_Water_Selective_Recover_Prev;
VO_Gas_Selective_Recover_Edge := VI_Gas_Selective_Recover AND NOT L_CMD_Gas_Selective_Recover_Prev;
VO_Water_Valve_Test_Open_Edge := VI_Water_Valve_Test_Open AND NOT L_CMD_Water_Valve_Test_Open_Prev;
VO_Water_Valve_Test_Close_Edge := VI_Water_Valve_Test_Close AND NOT L_CMD_Water_Valve_Test_Close_Prev;
VO_Water_Valve_Test_Confirm_Edge := VI_Water_Valve_Test_Confirm AND NOT L_CMD_Water_Valve_Test_Confirm_Prev;
VO_Gas_Valve_Test_Open_Edge := VI_Gas_Valve_Test_Open AND NOT L_CMD_Gas_Valve_Test_Open_Prev;
VO_Gas_Valve_Test_Close_Edge := VI_Gas_Valve_Test_Close AND NOT L_CMD_Gas_Valve_Test_Close_Prev;
VO_Gas_Valve_Test_Confirm_Edge := VI_Gas_Valve_Test_Confirm AND NOT L_CMD_Gas_Valve_Test_Confirm_Prev;

L_CMD_Water_Selective_Recover_Prev := VI_Water_Selective_Recover;
L_CMD_Gas_Selective_Recover_Prev := VI_Gas_Selective_Recover;
L_CMD_Water_Valve_Test_Open_Prev := VI_Water_Valve_Test_Open;
L_CMD_Water_Valve_Test_Close_Prev := VI_Water_Valve_Test_Close;
L_CMD_Water_Valve_Test_Confirm_Prev := VI_Water_Valve_Test_Confirm;
L_CMD_Gas_Valve_Test_Open_Prev := VI_Gas_Valve_Test_Open;
L_CMD_Gas_Valve_Test_Close_Prev := VI_Gas_Valve_Test_Close;
L_CMD_Gas_Valve_Test_Confirm_Prev := VI_Gas_Valve_Test_Confirm;

IF VO_Water_Valve_Test_Open_Edge THEN
    L_Water_Test_Active := TRUE;
    L_Water_Test_Deadline := VI_System_Time_MS + 60000;
END_IF;

IF L_Water_Test_Active THEN
    IF VI_System_Time_MS >= L_Water_Test_Deadline THEN
        L_Water_Test_Active := FALSE;
        VO_Water_Test_Timeout_Close_Required := TRUE;
    END_IF;
END_IF;

IF VO_Gas_Valve_Test_Open_Edge THEN
    L_Gas_Test_Active := TRUE;
    L_Gas_Test_Deadline := VI_System_Time_MS + 60000;
END_IF;

IF L_Gas_Test_Active THEN
    IF VI_System_Time_MS >= L_Gas_Test_Deadline THEN
        L_Gas_Test_Active := FALSE;
        VO_Gas_Test_Timeout_Close_Required := TRUE;
    END_IF;
END_IF;

VO_Water_Test_Active := L_Water_Test_Active;
VO_Gas_Test_Active := L_Gas_Test_Active;

(* ---- FB_State_Trace_Log.st ---- *)
FUNCTION_BLOCK FB_State_Trace_Log
VAR_INPUT
    VI_System_Time : UDINT;
    VI_Gas_Alarm : BOOL;
    VI_Leak_Alarm : BOOL;
    VI_Pumps : ARRAY[1..4] OF BOOL;
END_VAR
VAR_OUTPUT
    VO_Last_Change_Time : UDINT;
END_VAR
VAR
    L_Last_Gas : BOOL;
    L_Last_Leak : BOOL;
END_VAR

IF (VI_Gas_Alarm <> L_Last_Gas) OR (VI_Leak_Alarm <> L_Last_Leak) THEN
    VO_Last_Change_Time := VI_System_Time;
END_IF;

L_Last_Gas := VI_Gas_Alarm;
L_Last_Leak := VI_Leak_Alarm;

(* ---- FB_System_Timer_TOF.st ---- *)
// ==============================================================================
// Блок таймера задержки выключения (System Timer TOF)
// Назначение:
// - Замена стандартного TOF для обеспечения точной выдержки времени,
//   независимой от времени цикла ПЛК, с использованием единого системного времени.
// ==============================================================================
FUNCTION_BLOCK FB_System_Timer_TOF
VAR_INPUT
    IN : BOOL; // Вход запуска таймера
    PT : TIME; // Заданное время
    VI_System_Time_MS : UDINT; // Системное время (мс)
END_VAR
VAR_OUTPUT
    Q : BOOL; // Выход: таймер сработал
    ET : TIME; // Прошедшее время
END_VAR
VAR
    L_Start_Time : UDINT;
    L_Running : BOOL;
    L_Prev_IN : BOOL;
END_VAR

IF IN THEN
    Q := TRUE;
    ET := T#0s;
    L_Running := FALSE;
ELSE
    IF L_Prev_IN THEN
        L_Start_Time := VI_System_Time_MS;
        L_Running := TRUE;
        ET := T#0s;
    END_IF;

    IF L_Running THEN
        // Обработка переполнения UDINT (примерно 49 дней)
        ET := TO_TIME((SEL(VI_System_Time_MS >= L_Start_Time, VI_System_Time_MS - L_Start_Time, (4294967295 - L_Start_Time) + VI_System_Time_MS + 1)));

        IF ET >= PT THEN
            Q := FALSE;
            ET := PT;
            L_Running := FALSE;
        ELSE
            Q := TRUE;
        END_IF;
    END_IF;
END_IF;

L_Prev_IN := IN;

(* ---- PRG_IO_Read.st ---- *)
PROGRAM PRG_IO_Read
VAR
    L_i : INT;
    L_Debounce_Time : TIME := T#100MS;
    L_Manifold_Pressure_Raw : WORD;
    L_Manifold_Current_Raw : WORD;

    fbDebounce_Switches : ARRAY[1..8] OF FB_System_Timer;
    fbDebounce_Motion : ARRAY[1..8] OF FB_System_Timer;
    fbDebounce_Security_Open : ARRAY[1..GVL_CONSTANTS.C_MAX_SECURITY_SENSORS] OF FB_System_Timer;
    fbDebounce_Security_Glass : ARRAY[1..GVL_CONSTANTS.C_MAX_SECURITY_SENSORS] OF FB_System_Timer;
    fbDebounce_Flood : ARRAY[1..GVL_CONSTANTS.C_MAX_FLOOD_SENSORS] OF FB_System_Timer;
    fbDebounce_Smoke : ARRAY[1..GVL_CONSTANTS.C_MAX_SMOKE_SENSORS] OF FB_System_Timer;
    fbDebounce_Group_2F : FB_System_Timer;

    fbIO_Watchdog_1 : FB_IO_Module_Watchdog;
    fbIO_Watchdog_2 : FB_IO_Module_Watchdog;
    fbDiagEventManager : FB_Diagnostics_Event_Manager;
    L_IO_Error_Active : BOOL;

    // added
    fbCalib_Outdoor_Temp : FB_Sensor_Calibration_Processor;
    fbCalib_Supply_Temps : ARRAY[1..GVL_CONSTANTS.C_MAX_SUPPLY_TEMPS] OF FB_Sensor_Calibration_Processor;
    fbCalib_Room_Temps : ARRAY[1..GVL_CONSTANTS.C_MAX_ZONES] OF FB_Sensor_Calibration_Processor;
    fbCalib_Floor_Temps : ARRAY[1..GVL_CONSTANTS.C_MAX_ZONES] OF FB_Sensor_Calibration_Processor;
    fbCalib_Room_Hum : ARRAY[1..GVL_CONSTANTS.C_MAX_ZONES] OF FB_Sensor_Calibration_Processor;
    fbCalib_Room_CO2 : ARRAY[1..GVL_CONSTANTS.C_MAX_ZONES] OF FB_Sensor_Calibration_Processor;
    fbCalib_Manifold_T_Supply : ARRAY[1..GVL_CONSTANTS.C_MAX_MANIFOLDS] OF FB_Sensor_Calibration_Processor;
    fbCalib_Manifold_T_Return : ARRAY[1..GVL_CONSTANTS.C_MAX_MANIFOLDS] OF FB_Sensor_Calibration_Processor;
    fbCalib_Methane : ARRAY[1..GVL_CONSTANTS.C_MAX_METHANE_SENSORS] OF FB_Sensor_Calibration_Processor;
    fbCalib_CO : ARRAY[1..GVL_CONSTANTS.C_MAX_CO_SENSORS] OF FB_Sensor_Calibration_Processor;

    fbAnalog_Manifold_Pressure : ARRAY[1..GVL_CONSTANTS.C_MAX_MANIFOLDS] OF FB_Sensor_Analog_Processing;
    fbAnalog_Manifold_Current : ARRAY[1..GVL_CONSTANTS.C_MAX_MANIFOLDS] OF FB_Sensor_Analog_Processing;
END_VAR

// ===== ORIGINAL SNAPSHOT (FULL) =====
fbIO_Watchdog_1(VI_System_Time_MS := GVL_STATUS.G_System_Time_MS, VI_Module_ID := 1, VI_Heartbeat_Signal := GVL_IO.DI_Module_1_Heartbeat, VI_Timeout_MS := 2000);
fbIO_Watchdog_2(VI_System_Time_MS := GVL_STATUS.G_System_Time_MS, VI_Module_ID := 2, VI_Heartbeat_Signal := GVL_IO.DI_Module_2_Heartbeat, VI_Timeout_MS := 2000);

GVL_STATUS.G_IO_Modules_Online[1] := fbIO_Watchdog_1.VO_Module_Online;
GVL_STATUS.G_IO_Modules_Online[2] := fbIO_Watchdog_2.VO_Module_Online;

L_IO_Error_Active := fbIO_Watchdog_1.VO_Error_Active OR fbIO_Watchdog_2.VO_Error_Active;

// IO watchdog events
fbDiagEventManager(
    VI_Code := 16#E001,
    VI_Severity := 4,
    VI_Active := NOT fbIO_Watchdog_1.VO_Module_Online,
    VI_Timestamp := GVL_STATUS.G_System_Time_MS,
    VI_Source := 1,
    VIO_Events := GVL_STATUS.G_Diagnostics_Events,
    VIO_Count := GVL_STATUS.G_Diagnostics_Count
);

fbDiagEventManager(
    VI_Code := 16#E002,
    VI_Severity := 4,
    VI_Active := NOT fbIO_Watchdog_2.VO_Module_Online,
    VI_Timestamp := GVL_STATUS.G_System_Time_MS,
    VI_Source := 2,
    VIO_Events := GVL_STATUS.G_Diagnostics_Events,
    VIO_Count := GVL_STATUS.G_Diagnostics_Count
);

IF L_IO_Error_Active THEN
    GVL_COMMAND.G_Gas_Valve_Close := TRUE;
    GVL_COMMAND.G_Close_Valve_35 := TRUE;
    GVL_COMMAND.G_Close_Valve_36 := TRUE;
    FOR L_i := 1 TO GVL_CONSTANTS.C_MAX_MANIFOLDS DO GVL_STATE.G_Manifold_Pumps[L_i] := FALSE; END_FOR;
END_IF;

FOR L_i := 1 TO 8 DO
    fbDebounce_Switches[L_i](IN := GVL_IO.DI_Lighting_Switches[L_i], PT := L_Debounce_Time, VI_System_Time_MS := GVL_STATUS.G_System_Time_MS);
    GVL_STATE.G_Physical_Switches[L_i] := fbDebounce_Switches[L_i].Q;

    fbDebounce_Motion[L_i](IN := GVL_IO.DI_Motion_Sensors[L_i], PT := L_Debounce_Time, VI_System_Time_MS := GVL_STATUS.G_System_Time_MS);
    GVL_STATE.G_Motion_Sensors[L_i] := fbDebounce_Motion[L_i].Q;
END_FOR;

FOR L_i := 1 TO GVL_CONSTANTS.C_MAX_SOCKETS DO
    GVL_STATE.G_Socket_Switches[L_i] := FALSE;
END_FOR;

FOR L_i := 1 TO GVL_CONSTANTS.C_MAX_SECURITY_SENSORS DO
    fbDebounce_Security_Open[L_i](IN := GVL_IO.DI_Security_Open[L_i], PT := L_Debounce_Time, VI_System_Time_MS := GVL_STATUS.G_System_Time_MS);
    fbDebounce_Security_Glass[L_i](IN := GVL_IO.DI_Security_Glass[L_i], PT := L_Debounce_Time, VI_System_Time_MS := GVL_STATUS.G_System_Time_MS);
END_FOR;

fbDebounce_Group_2F(IN := GVL_IO.DI_Security_2F_Group, PT := L_Debounce_Time, VI_System_Time_MS := GVL_STATUS.G_System_Time_MS);

FOR L_i := 1 TO GVL_CONSTANTS.C_MAX_DOOR_SENSORS DO
    IF GVL_CONFIG.G_Door_Map[L_i] > 0 AND GVL_CONFIG.G_Door_Map[L_i] <= GVL_CONSTANTS.C_MAX_SECURITY_SENSORS THEN
        GVL_STATE.G_Door_Sensors[L_i] := fbDebounce_Security_Open[GVL_CONFIG.G_Door_Map[L_i]].Q;
    END_IF;
END_FOR;

FOR L_i := 1 TO 8 DO
    IF GVL_CONFIG.G_Window_Map[L_i] > 0 THEN
        IF GVL_CONFIG.G_Window_Map[L_i] <= GVL_CONSTANTS.C_MAX_SECURITY_SENSORS THEN
            GVL_STATE.G_Window_Sensors[L_i] := fbDebounce_Security_Open[GVL_CONFIG.G_Window_Map[L_i]].Q;
        ELSE
            GVL_STATE.G_Window_Sensors[L_i] := fbDebounce_Security_Glass[GVL_CONFIG.G_Window_Map[L_i] - GVL_CONSTANTS.C_MAX_SECURITY_SENSORS].Q;
        END_IF;
    END_IF;
END_FOR;
GVL_STATE.G_Window_Sensors[16] := fbDebounce_Group_2F.Q;

FOR L_i := 1 TO GVL_CONSTANTS.C_MAX_FLOOD_SENSORS DO
    fbDebounce_Flood[L_i](IN := GVL_IO.DI_Flood_Sensors[L_i], PT := L_Debounce_Time, VI_System_Time_MS := GVL_STATUS.G_System_Time_MS);
    GVL_STATE.G_Water_Sensors[L_i] := fbDebounce_Flood[L_i].Q;
END_FOR;

FOR L_i := 1 TO GVL_CONSTANTS.C_MAX_SMOKE_SENSORS DO
    fbDebounce_Smoke[L_i](IN := GVL_IO.DI_Smoke_Sensors[L_i], PT := L_Debounce_Time, VI_System_Time_MS := GVL_STATUS.G_System_Time_MS);
    GVL_STATE.G_Smoke_Sensors[L_i] := fbDebounce_Smoke[L_i].Q;
END_FOR;

// ===== ENHANCED LAYER =====
fbCalib_Outdoor_Temp(
    VI_Raw_Value := GVL_IO.AI_Temp_Outdoor.rValue,
    VI_Record := GVL_CONFIG.G_Calib_Outdoor_Temp
);
GVL_STATE.G_Outdoor_Temp := fbCalib_Outdoor_Temp.VO_Calibrated_Value;

FOR L_i := 1 TO GVL_CONSTANTS.C_MAX_SUPPLY_TEMPS DO
    IF GVL_IO.AI_Supply_Temps[L_i].wStatus = 0 THEN
        fbCalib_Supply_Temps[L_i](
            VI_Raw_Value := GVL_IO.AI_Supply_Temps[L_i].rValue,
            VI_Record := GVL_CONFIG.G_Calib_Supply_Temps[L_i]
        );
        GVL_STATE.G_Supply_Temps[L_i] := fbCalib_Supply_Temps[L_i].VO_Calibrated_Value;
    END_IF;
END_FOR;

FOR L_i := 1 TO 8 DO
    fbCalib_Room_Hum[L_i](
        VI_Raw_Value := GVL_IO.AI_Room_Hum[L_i],
        VI_Record := GVL_CONFIG.G_Calib_Humidity[L_i]
    );
    GVL_STATE.G_Room_Hum[L_i] := fbCalib_Room_Hum[L_i].VO_Calibrated_Value;

    fbCalib_Room_CO2[L_i](
        VI_Raw_Value := GVL_IO.AI_Room_CO2[L_i],
        VI_Record := GVL_CONFIG.G_Calib_CO2[L_i]
    );
    GVL_STATE.G_Room_CO2[L_i] := fbCalib_Room_CO2[L_i].VO_Calibrated_Value;
END_FOR;

FOR L_i := 1 TO 8 DO
    fbCalib_Room_Temps[L_i](
        VI_Raw_Value := GVL_IO.AI_Room_Temps[L_i],
        VI_Record := GVL_CONFIG.G_Calib_Room_Temps[L_i]
    );
    GVL_STATE.G_Room_Temps[L_i] := fbCalib_Room_Temps[L_i].VO_Calibrated_Value;

    fbCalib_Floor_Temps[L_i](
        VI_Raw_Value := GVL_IO.AI_Floor_Temps[L_i],
        VI_Record := GVL_CONFIG.G_Calib_Floor_Temps[L_i]
    );
    GVL_STATE.G_Floor_Temps[L_i] := fbCalib_Floor_Temps[L_i].VO_Calibrated_Value;
END_FOR;

GVL_STATUS.G_Diagnostics.Manifold_Pressure_Fault_Active := FALSE;
GVL_STATUS.G_Diagnostics.Manifold_Pressure_First_Fault_Index := 0;
GVL_STATUS.G_Diagnostics.Manifold_Current_Fault_Active := FALSE;
GVL_STATUS.G_Diagnostics.Manifold_Current_First_Fault_Index := 0;
GVL_STATUS.G_Diagnostics.Manifold_Pressure_Fault_Text := '';
GVL_STATUS.G_Diagnostics.Manifold_Current_Fault_Text := '';
GVL_STATUS.G_Diagnostics.Sensor_Fault := FALSE;
GVL_STATUS.G_Diagnostics.Subsystem_Degraded := FALSE;

FOR L_i := 1 TO GVL_CONSTANTS.C_MAX_MANIFOLDS DO
    IF GVL_IO.AI_Manifold_Pressures[L_i] < 0 THEN
        L_Manifold_Pressure_Raw := 0;
    ELSE
        L_Manifold_Pressure_Raw := INT_TO_WORD(GVL_IO.AI_Manifold_Pressures[L_i]);
    END_IF;

    IF GVL_IO.AI_Manifold_Currents[L_i] < 0 THEN
        L_Manifold_Current_Raw := 0;
    ELSE
        L_Manifold_Current_Raw := INT_TO_WORD(GVL_IO.AI_Manifold_Currents[L_i]);
    END_IF;

    fbAnalog_Manifold_Pressure[L_i](
        VI_Raw_Value := L_Manifold_Pressure_Raw,
        VI_Sensor_Type := 0,
        VI_Min_Scale := 0.0,
        VI_Max_Scale := 10.0,
        VI_Offset := 0.0,
        VI_Multiplier := 1.0,
        VI_Filter_Time_MS := GVL_CONSTANTS.C_MS_IN_SECOND,
        VI_System_Time_MS := GVL_STATUS.G_System_Time_MS,
        VI_Fallback_Mode := 0,
        VI_Default_Value := 0.0
    );
    GVL_STATE.G_Manifold_Pressures[L_i] := fbAnalog_Manifold_Pressure[L_i].VO_Value;
    GVL_STATUS.G_Diagnostics.Manifold_Pressure_Fault[L_i] := fbAnalog_Manifold_Pressure[L_i].VO_Error;
    GVL_STATUS.G_Diagnostics.Manifold_Pressure_Diag_Code[L_i] := fbAnalog_Manifold_Pressure[L_i].VO_Diag_Code;

    fbDiagEventManager(
        VI_Code := GVL_CONFIG.ERR_PRESSURE_OUT_OF_RANGE,
        VI_Severity := 3,
        VI_Active := fbAnalog_Manifold_Pressure[L_i].VO_Error,
        VI_Timestamp := GVL_STATUS.G_System_Time_MS,
        VI_Source := 100 + L_i,
        VIO_Events := GVL_STATUS.G_Diagnostics_Events,
        VIO_Count := GVL_STATUS.G_Diagnostics_Count
    );

    fbAnalog_Manifold_Current[L_i](
        VI_Raw_Value := L_Manifold_Current_Raw,
        VI_Sensor_Type := 0,
        VI_Min_Scale := 0.0,
        VI_Max_Scale := 16.0,
        VI_Offset := 0.0,
        VI_Multiplier := 1.0,
        VI_Filter_Time_MS := GVL_CONSTANTS.C_MS_IN_SECOND,
        VI_System_Time_MS := GVL_STATUS.G_System_Time_MS,
        VI_Fallback_Mode := 0,
        VI_Default_Value := 0.0
    );
    GVL_STATE.G_Manifold_Currents[L_i] := fbAnalog_Manifold_Current[L_i].VO_Value;
    GVL_STATUS.G_Diagnostics.Manifold_Current_Fault[L_i] := fbAnalog_Manifold_Current[L_i].VO_Error;
    GVL_STATUS.G_Diagnostics.Manifold_Current_Diag_Code[L_i] := fbAnalog_Manifold_Current[L_i].VO_Diag_Code;

    fbDiagEventManager(
        VI_Code := GVL_CONFIG.ERR_PUMP_UNDERCURRENT,
        VI_Severity := 3,
        VI_Active := fbAnalog_Manifold_Current[L_i].VO_Error,
        VI_Timestamp := GVL_STATUS.G_System_Time_MS,
        VI_Source := 200 + L_i,
        VIO_Events := GVL_STATUS.G_Diagnostics_Events,
        VIO_Count := GVL_STATUS.G_Diagnostics_Count
    );

    IF GVL_IO.AI_Manifold_Temps_Supply[L_i].wStatus = 0 THEN
        fbCalib_Manifold_T_Supply[L_i](
            VI_Raw_Value := GVL_IO.AI_Manifold_Temps_Supply[L_i].rValue,
            VI_Record := GVL_CONFIG.G_Calib_Manifold_T_Supply[L_i]
        );
        GVL_STATE.G_Manifold_T_Supply[L_i] := fbCalib_Manifold_T_Supply[L_i].VO_Calibrated_Value;
    END_IF;

    fbCalib_Manifold_T_Return[L_i](
        VI_Raw_Value := INT_TO_REAL(GVL_IO.AI_Manifold_Temps_Return[L_i]) / 10.0,
        VI_Record := GVL_CONFIG.G_Calib_Manifold_T_Return[L_i]
    );
    GVL_STATE.G_Manifold_T_Return[L_i] := fbCalib_Manifold_T_Return[L_i].VO_Calibrated_Value;
    GVL_STATE.G_Manifold_End_Switches[L_i] := GVL_IO.DI_Manifold_End_Switches[L_i];

    IF GVL_STATUS.G_Diagnostics.Manifold_Pressure_Fault[L_i] OR GVL_STATUS.G_Diagnostics.Manifold_Current_Fault[L_i] THEN
        GVL_STATUS.G_Diagnostics.Sensor_Fault := TRUE;
        GVL_STATUS.G_Diagnostics.Subsystem_Degraded := TRUE;
    END_IF;

    IF GVL_STATUS.G_Diagnostics.Manifold_Pressure_Fault[L_i] AND GVL_STATUS.G_Diagnostics.Manifold_Current_Fault[L_i] THEN
        GVL_STATUS.G_Diagnostics.Manifold_Pressure_Fault_Text := 'Correlated pressure/current fault detected';
        GVL_STATUS.G_Diagnostics.Manifold_Current_Fault_Text := 'Correlated pressure/current fault detected';
    ELSIF GVL_STATUS.G_Diagnostics.Manifold_Pressure_Fault[L_i] AND (GVL_STATUS.G_Diagnostics.Manifold_Pressure_Fault_Text = '') THEN
        GVL_STATUS.G_Diagnostics.Manifold_Pressure_Fault_Text := 'Pressure sensor fault detected';
    ELSIF GVL_STATUS.G_Diagnostics.Manifold_Current_Fault[L_i] AND (GVL_STATUS.G_Diagnostics.Manifold_Current_Fault_Text = '') THEN
        GVL_STATUS.G_Diagnostics.Manifold_Current_Fault_Text := 'Current sensor fault detected';
    END_IF;
END_FOR;

FOR L_i := 1 TO GVL_CONSTANTS.C_MAX_METHANE_SENSORS DO
    IF GVL_IO.AI_Methane_LEL[L_i].wStatus = 0 THEN
        fbCalib_Methane[L_i](
            VI_Raw_Value := GVL_IO.AI_Methane_LEL[L_i].rValue,
            VI_Record := GVL_CONFIG.G_Calib_Methane[L_i]
        );
        GVL_STATE.G_Methane_Sensors[L_i] := fbCalib_Methane[L_i].VO_Calibrated_Value;
    END_IF;

    fbDiagEventManager(
        VI_Code := 16#E003,
        VI_Severity := 3,
        VI_Active := GVL_IO.AI_Methane_LEL[L_i].wStatus <> 0,
        VI_Timestamp := GVL_STATUS.G_System_Time_MS,
        VI_Source := 300 + L_i,
        VIO_Events := GVL_STATUS.G_Diagnostics_Events,
        VIO_Count := GVL_STATUS.G_Diagnostics_Count
    );
END_FOR;

FOR L_i := 1 TO GVL_CONSTANTS.C_MAX_CO_SENSORS DO
    fbCalib_CO[L_i](
        VI_Raw_Value := GVL_IO.AI_CO_PPM[L_i],
        VI_Record := GVL_CONFIG.G_Calib_CO[L_i]
    );
    GVL_STATE.G_CO_Sensors[L_i] := fbCalib_CO[L_i].VO_Calibrated_Value;
END_FOR;

GVL_STATE.G_Boiler_Flame := GVL_IO.AI_Boiler_Flame_Status;
GVL_STATE.G_Boiler_Error := GVL_IO.DI_Boiler_Error;
FOR L_i := 1 TO GVL_CONSTANTS.C_MAX_BOILERS DO
    GVL_STATE.G_Boiler_OT_Online[L_i] := FALSE;
END_FOR;

GVL_STATE.G_DHW_Temp := GVL_IO.AI_DHW_Temp;
GVL_STATE.G_DHW_Pressure := GVL_IO.AI_DHW_Pressure;

GVL_STATE.G_Water_Zone_Open_FB := GVL_IO.DI_Water_Zone_Open_FB;
GVL_STATE.G_Water_Zone_Close_FB := GVL_IO.DI_Water_Zone_Close_FB;

// >>> BULK_SYNC_ANCHOR: PRG_IO_Read <<<

(* ---- PRG_IO_Write.st ---- *)
PROGRAM PRG_IO_Write
VAR
    L_i : INT;
END_VAR

// 2. ЗАПИСЬ ВЫХОДОВ (GVL_STATE -> GVL_IO)

// 2.1. Отопление (Термоэлектрические приводы)
FOR L_i := 1 TO 8 DO
    GVL_IO.DO_Zone_Valves[L_i] := GVL_STATE.G_Zone_Valves[L_i];
END_FOR;

// 2.2. Коллекторы (Насосы и смесительные клапаны)
FOR L_i := 1 TO GVL_CONSTANTS.C_MAX_MANIFOLDS DO
    GVL_IO.DO_Manifold_Pumps[L_i] := GVL_STATE.G_Manifold_Pumps[L_i];
    GVL_IO.AO_Manifold_Valves[L_i] := REAL_TO_UINT(GVL_STATE.G_Manifold_Valves[L_i] * 1000.0);
END_FOR;

// 2.4. Вентиляция
FOR L_i := 1 TO GVL_CONSTANTS.C_MAX_SUPPLY_FANS DO
    GVL_IO.AO_Supply_Fans[L_i] := REAL_TO_UINT(GVL_STATE.G_Supply_Fans[L_i] * 100.0);
END_FOR;
FOR L_i := 1 TO GVL_CONSTANTS.C_MAX_EXHAUST_FANS DO
    GVL_IO.AO_Exhaust_Fans[L_i] := REAL_TO_UINT(GVL_STATE.G_Exhaust_Fans[L_i] * 100.0);
END_FOR;

// 2.5. ГВС
GVL_IO.DO_DHW_Heating_Pump := GVL_STATE.G_DHW_Heating_Pump;
GVL_IO.DO_DHW_Circ_Pump := GVL_STATE.G_DHW_Circ_Pump;
IF GVL_STATUS.G_Is_Active_PLC THEN
    GVL_IO.DO_Backup_Circulation_Pump := GVL_STATE.G_Backup_Circulation_Pump;
    GVL_IO.DO_Electric_Heater_Enable := GVL_STATE.G_Electric_Heater_Enable;
ELSE
    GVL_IO.DO_Backup_Circulation_Pump := FALSE;
    GVL_IO.DO_Electric_Heater_Enable := FALSE;
END_IF;

// 2.6. Освещение и шторы
FOR L_i := 1 TO 8 DO
    GVL_IO.AO_Lighting_Levels[L_i] := BYTE_TO_UINT(GVL_STATE.G_Lighting_Levels[L_i]) * 10;
END_FOR;
FOR L_i := 1 TO GVL_CONSTANTS.C_MAX_BLINDS DO
    GVL_IO.AO_Blinds_Positions[L_i] := BYTE_TO_UINT(GVL_STATE.G_Blinds_Positions[L_i]) * 10;
END_FOR;

// 2.7. Аварийные выходы (Сирены и клапаны)
GVL_IO.DO_Gas_Siren := (GVL_ALARM.G_Gas_Fire_Siren AND GVL_ALARM.G_Gas_Alarm_Active);
GVL_IO.DO_Fire_Siren := (GVL_ALARM.G_Gas_Fire_Siren AND GVL_ALARM.G_Fire_Alarm_Active);
GVL_IO.DO_Security_Siren := GVL_ALARM.G_Security_Siren;

// === STAGE H2: USE SHADOW COMMANDS ===
GVL_IO.DO_Water_Valve_35_Close := GVL_COMMAND_SHADOW.G_Close_Valve_35;
GVL_IO.DO_Water_Valve_36_Close := GVL_COMMAND_SHADOW.G_Close_Valve_36;
GVL_IO.DO_Gas_Valve_Close := GVL_COMMAND_SHADOW.G_Gas_Valve_Close;

// Access control (shadow)
GVL_IO.DO_Lock_1_Open := GVL_COMMAND_SHADOW.G_Lock_1_Open;
GVL_IO.DO_Lock_1_Close := GVL_COMMAND_SHADOW.G_Lock_1_Close;
GVL_IO.DO_Lock_2_Open := GVL_COMMAND_SHADOW.G_Lock_2_Open;
GVL_IO.DO_Lock_2_Close := GVL_COMMAND_SHADOW.G_Lock_2_Close;

// Gate/Wicket — now via shadow
GVL_IO.DO_Gate_Open := GVL_COMMAND_SHADOW.G_Gate_Open;
GVL_IO.DO_Wicket_Open := GVL_COMMAND_SHADOW.G_Wicket_Open;

// 2.9. Розетки
GVL_IO.DO_Sockets := GVL_STATE.G_Socket_States;

// Selective zonal water recovery outputs
FOR L_i := 1 TO 32 DO
    GVL_IO.DO_Water_Zone_Enable[L_i] := GVL_STATE.G_Water_Zone_Enable[L_i];
END_FOR;

// >>> BULK_SYNC_ANCHOR: PRG_IO_Write <<<

(* ---- PRG_Lighting.st ---- *)
PROGRAM PRG_Lighting
VAR
    L_i : INT;
    fbLightingManager : FB_Lighting_Blinds_Manager;
    fbSocketManager : FB_Socket_Manager;
    L_Manual_Light_Override_32 : ARRAY[1..32] OF BYTE;
    L_Manual_Blinds_Override_32 : ARRAY[1..32] OF BYTE;
    L_Manual_Socket_Override_32 : ARRAY[1..32] OF BOOL;
    L_Sim_Lights_32 : ARRAY[1..32] OF BOOL;
    L_Physical_Switches_32 : ARRAY[1..32] OF BOOL;
    L_Motion_Sensors_32 : ARRAY[1..32] OF BOOL;

    // ADAPTER ARRAYS (match FB expected sizes)
    L_Blinds_Override : ARRAY[1..GVL_CONSTANTS.C_MAX_BLINDS] OF BYTE;
    L_Socket_Override : ARRAY[1..GVL_CONSTANTS.C_MAX_SOCKETS] OF BOOL;
END_VAR

FOR L_i := 1 TO 32 DO
    IF L_i <= 16 THEN
        IF GVL_INTENT_SYSTEM.I_Lighting_Overrides_Block OR GVL_SYSTEM_COORDINATION.G_Block_Lighting_Override THEN
            L_Manual_Light_Override_32[L_i] := 0;
        ELSE
            L_Manual_Light_Override_32[L_i] := GVL_INTENT_USER.I_Lighting_Override_32[L_i];
        END_IF;
        L_Sim_Lights_32[L_i] := GVL_STATE.G_Sim_Lights[L_i];
        L_Physical_Switches_32[L_i] := GVL_STATE.G_Physical_Switches[L_i];
        L_Motion_Sensors_32[L_i] := GVL_STATE.G_Motion_Sensors[L_i];
    ELSE
        L_Manual_Light_Override_32[L_i] := 0;
        L_Sim_Lights_32[L_i] := FALSE;
        L_Physical_Switches_32[L_i] := FALSE;
        L_Motion_Sensors_32[L_i] := FALSE;
    END_IF;

    IF GVL_INTENT_SYSTEM.I_Blinds_Overrides_Block THEN
        L_Manual_Blinds_Override_32[L_i] := 0;
    ELSE
        L_Manual_Blinds_Override_32[L_i] := GVL_INTENT_USER.I_Blinds_Override_32[L_i];
    END_IF;

    IF GVL_INTENT_SYSTEM.I_Socket_Overrides_Block OR GVL_SYSTEM_COORDINATION.G_Block_Sockets_Override THEN
        L_Manual_Socket_Override_32[L_i] := FALSE;
    ELSE
        L_Manual_Socket_Override_32[L_i] := GVL_INTENT_USER.I_Socket_Override_32[L_i];
    END_IF;
END_FOR;

// ADAPTER: copy to FB-sized arrays
FOR L_i := 1 TO GVL_CONSTANTS.C_MAX_BLINDS DO
    L_Blinds_Override[L_i] := L_Manual_Blinds_Override_32[L_i];
END_FOR;

FOR L_i := 1 TO GVL_CONSTANTS.C_MAX_SOCKETS DO
    L_Socket_Override[L_i] := L_Manual_Socket_Override_32[L_i];
END_FOR;

// 10. Управление освещением и шторами
fbLightingManager(
    VI_System_Time_MS := GVL_STATUS.G_System_Time_MS,
    VI_IsActivePLC := GVL_STATUS.G_Is_Active_PLC,
    VI_Current_Scenario := GVL_STATUS.G_Current_Scenario,
    VI_Away_Level := 1,
    VI_Simulation_Active := GVL_STATUS.G_Sim_Active,
    VI_Manual_Light_Override := L_Manual_Light_Override_32,
    VI_Manual_Blinds_Override := L_Blinds_Override,
    VI_Simulation_Lights := L_Sim_Lights_32,
    VI_Physical_Switches := L_Physical_Switches_32,
    VI_Motion_Sensors := L_Motion_Sensors_32,
    VI_Is_Night := GVL_STATUS.G_Is_Night,
    VI_Rule_Actions := GVL_STATE.G_Rule_Actions,
    VI_IO_Modules_Online := GVL_STATUS.G_IO_Modules_Online,
    VI_Wet_Zone_Map := GVL_CONFIG.G_Wet_Zone_Map,
    VI_Scenario_Configs := GVL_CONFIG.G_HMI_Scenario_Configs,
    VO_Lighting_Levels => GVL_STATE.G_Lighting_Levels,
    VO_Blinds_Positions => GVL_STATE.G_Blinds_Positions
);

// 11.5 Управление розетками
fbSocketManager(
    VI_System_Time_MS := GVL_STATUS.G_System_Time_MS,
    VI_IsActivePLC := GVL_STATUS.G_Is_Active_PLC,
    VI_Scenario := GVL_STATUS.G_Current_Scenario,
    VI_Manual_Override := L_Socket_Override,
    VI_Physical_Switches := GVL_STATE.G_Socket_Switches,
    VI_Rule_Actions := GVL_STATE.G_Rule_Actions,
    VI_Fire_Alarm := GVL_ALARM.G_Fire_Alarm_Active,
    VI_Flood_Alarm := GVL_ALARM.G_Flood_Alarm_Active,
    VI_Security_Armed := GVL_ALARM.G_Security_Armed,
    VI_IO_Modules_Online := GVL_STATUS.G_IO_Modules_Online,
    VO_Socket_States => GVL_STATE.G_Socket_States
);

// Evacuation lighting override
IF GVL_STATE.G_Evacuation_Lighting_Active THEN
    FOR L_i := 1 TO 8 DO
        IF (L_i MOD 2) = 0 THEN
            GVL_STATE.G_Lighting_Levels[L_i] := 100;
        ELSE
            GVL_STATE.G_Lighting_Levels[L_i] := 0;
        END_IF;
    END_FOR;
END_IF;

// Directional evacuation override
IF GVL_STATE.G_Evacuation_Lighting_Active THEN
    FOR L_i := 1 TO GVL_CONFIG.C_MAX_LIGHT_ZONES DO
        CASE GVL_STATE.G_Evac_Guidance[L_i] OF
            -1:
                GVL_STATE.G_Lighting_Levels[L_i] := 0;
            1:
                GVL_STATE.G_Lighting_Levels[L_i] := 100;
        ELSE
            GVL_STATE.G_Lighting_Levels[L_i] := SEL((L_i MOD 2) = 0, 0, 100);
        END_CASE;
    END_FOR;
END_IF;
// >>> BULK_SYNC_ANCHOR: PRG_Lighting <<<

(* ---- PRG_Presence_Manager.st ---- *)
PROGRAM PRG_Presence_Manager
VAR
    fbPresence : FB_Presence_Manager;
    L_i : INT;
END_VAR

fbPresence(
    VI_Motion_Sensors := GVL_STATE.G_Motion_Sensors,
    VI_System_Time_MS := GVL_STATUS.G_System_Time_MS
);

GVL_PRESENCE.G_Any_Motion := fbPresence.VO_Any_Motion;
GVL_PRESENCE.G_Occupied := fbPresence.VO_Occupied;
GVL_PRESENCE.G_Auto_Away_Request := fbPresence.VO_Auto_Away;
GVL_PRESENCE.G_Last_Motion_TS := fbPresence.VO_Last_Motion_TS;

FOR L_i := 1 TO GVL_CONSTANTS.C_MAX_ZONES DO
    IF GVL_STATE.G_Motion_Sensors[L_i] THEN
        GVL_PRESENCE.G_Zone_Occupied[L_i] := TRUE;
        GVL_PRESENCE.G_Zone_Last_Motion_TS[L_i] := GVL_STATUS.G_System_Time_MS;
    END_IF;

    IF (GVL_STATUS.G_System_Time_MS - GVL_PRESENCE.G_Zone_Last_Motion_TS[L_i]) > 900000 THEN
        GVL_PRESENCE.G_Zone_Occupied[L_i] := FALSE;
    END_IF;
END_FOR;

(* ---- PRG_System_Test_Harness.st ---- *)
PROGRAM PRG_System_Test_Harness
VAR
    L_i : INT;
    L_j : INT;
    L_Used : REAL;
    L_HP_Used : REAL;
    L_HP_Manifold_Adjusted : ARRAY[1..GVL_CONSTANTS.C_MAX_MANIFOLDS] OF INT;
    fbDecisionTest : FB_Heating_Decision_Context;
    fbDecisionHP : FB_Heating_Decision_Context;
    fbTestResult : FB_Test_Result_Handler;
    fbTrace : FB_Trace_Logger;
END_VAR

IF NOT GVL_TEST.G_Test_Enable THEN
    RETURN;
END_IF;

GVL_TEST.G_Test_Total_Checks := 0;
GVL_TEST.G_Test_Failed_Checks := 0;
GVL_TEST.G_Test_Passed := TRUE;
GVL_TEST.G_Test_Last_Failure_Index := 0;
GVL_TEST.G_Test_Last_Failure_Code := 0;

// Reset transient failure flags for this scan
GVL_TEST.G_Diagnostics_Duplicate_Event_Found := FALSE;
GVL_TEST.G_Diagnostics_Count_Out_Of_Range := FALSE;
GVL_TEST.G_Heating_Allocation_Budget_Exceeded := FALSE;
GVL_TEST.G_Heating_Allocation_Enabled_Not_Allowed := FALSE;
GVL_TEST.G_Safety_Latched_Without_Intent := FALSE;
GVL_TEST.G_HP_Adjusted_Priority_Lower_Bound_Violation := FALSE;
GVL_TEST.G_HP_Adjusted_Allocation_Budget_Exceeded := FALSE;
GVL_TEST.G_HP_Adjusted_Allocation_Enabled_Not_Allowed := FALSE;
GVL_TEST.G_HP_Guest_Preheat_Config_Out_Of_Range := FALSE;

// =========================
// TEST 1: Diagnostics count bounds
// =========================
GVL_TEST.G_Test_Total_Checks := GVL_TEST.G_Test_Total_Checks + 1;
IF (GVL_STATUS.G_Diagnostics_Count < 0) OR (GVL_STATUS.G_Diagnostics_Count > 50) THEN
    GVL_TEST.G_Diagnostics_Count_Out_Of_Range := TRUE;
    GVL_TEST.G_Test_Failed_Checks := GVL_TEST.G_Test_Failed_Checks + 1;
    GVL_TEST.G_Test_Passed := FALSE;
    GVL_TEST.G_Test_Last_Failure_Index := 1;
    GVL_TEST.G_Test_Last_Failure_Code := 1001;
END_IF;

// =========================
// TEST 2: Diagnostics duplicates
// =========================
GVL_TEST.G_Test_Total_Checks := GVL_TEST.G_Test_Total_Checks + 1;
FOR L_i := 1 TO GVL_STATUS.G_Diagnostics_Count DO
    FOR L_j := L_i + 1 TO GVL_STATUS.G_Diagnostics_Count DO
        IF (GVL_STATUS.G_Diagnostics_Events[L_i].Code = GVL_STATUS.G_Diagnostics_Events[L_j].Code) AND
           (GVL_STATUS.G_Diagnostics_Events[L_i].Source = GVL_STATUS.G_Diagnostics_Events[L_j].Source) THEN
            GVL_TEST.G_Diagnostics_Duplicate_Event_Found := TRUE;
            GVL_TEST.G_Test_Failed_Checks := GVL_TEST.G_Test_Failed_Checks + 1;
            GVL_TEST.G_Test_Passed := FALSE;
            GVL_TEST.G_Test_Last_Failure_Index := 2;
            GVL_TEST.G_Test_Last_Failure_Code := 1002;
        END_IF;
    END_FOR;
END_FOR;

// =========================
// TEST 3: Base heating decision consistency
// =========================
GVL_TEST.G_Test_Total_Checks := GVL_TEST.G_Test_Total_Checks + 1;
fbDecisionTest(
    VI_Manifold_Pump_In_Service := GVL_CONFIG.G_Manifold_Pump_In_Service,
    VI_Manifold_Pressure_Fault := GVL_STATUS.G_Diagnostics.Manifold_Pressure_Fault,
    VI_Manifold_Current_Fault := GVL_STATUS.G_Diagnostics.Manifold_Current_Fault,
    VI_Manifold_Thermal_Weight := GVL_CONFIG.G_Manifold_Thermal_Weight,
    VI_Manifold_Priority := GVL_CONFIG.G_Manifold_Priority,
    VI_Max_Thermal_Budget := GVL_CONFIG.G_Max_Thermal_Budget
);

L_Used := 0.0;
FOR L_i := 1 TO GVL_CONSTANTS.C_MAX_MANIFOLDS DO
    IF fbDecisionTest.VO_Manifold_Enabled[L_i] AND (NOT fbDecisionTest.VO_Manifold_Allowed[L_i]) THEN
        GVL_TEST.G_Heating_Allocation_Enabled_Not_Allowed := TRUE;
        GVL_TEST.G_Test_Failed_Checks := GVL_TEST.G_Test_Failed_Checks + 1;
        GVL_TEST.G_Test_Passed := FALSE;
        GVL_TEST.G_Test_Last_Failure_Index := 3;
        GVL_TEST.G_Test_Last_Failure_Code := 1003;
    END_IF;

    IF fbDecisionTest.VO_Manifold_Enabled[L_i] THEN
        L_Used := L_Used + GVL_CONFIG.G_Manifold_Thermal_Weight[L_i];
    END_IF;
END_FOR;

IF L_Used > (GVL_CONFIG.G_Max_Thermal_Budget + 0.001) THEN
    GVL_TEST.G_Heating_Allocation_Budget_Exceeded := TRUE;
    GVL_TEST.G_Test_Failed_Checks := GVL_TEST.G_Test_Failed_Checks + 1;
    GVL_TEST.G_Test_Passed := FALSE;
    GVL_TEST.G_Test_Last_Failure_Index := 3;
    GVL_TEST.G_Test_Last_Failure_Code := 1004;
END_IF;

// =========================
// TEST 4: Safety latch consistency
// =========================
GVL_TEST.G_Test_Total_Checks := GVL_TEST.G_Test_Total_Checks + 1;
IF GVL_STATE.G_Safety_Gas_Latched AND (NOT GVL_INTENT_SAFETY.I_Gas_Alarm_Active) THEN
    GVL_TEST.G_Safety_Latched_Without_Intent := TRUE;
    GVL_TEST.G_Test_Failed_Checks := GVL_TEST.G_Test_Failed_Checks + 1;
    GVL_TEST.G_Test_Passed := FALSE;
    GVL_TEST.G_Test_Last_Failure_Index := 4;
    GVL_TEST.G_Test_Last_Failure_Code := 1005;
END_IF;

// =========================
// TEST 5: HP policy adjusted priority
// =========================
GVL_TEST.G_Test_Total_Checks := GVL_TEST.G_Test_Total_Checks + 1;

IF (GVL_HEATING_POLICY_CONFIG.G_Guest_Preheat_Priority_Boost < 0) OR (GVL_HEATING_POLICY_CONFIG.G_Guest_Preheat_Priority_Boost > 10) THEN
    GVL_TEST.G_HP_Guest_Preheat_Config_Out_Of_Range := TRUE;
    GVL_TEST.G_Test_Failed_Checks := GVL_TEST.G_Test_Failed_Checks + 1;
    GVL_TEST.G_Test_Passed := FALSE;
    GVL_TEST.G_Test_Last_Failure_Index := 5;
    GVL_TEST.G_Test_Last_Failure_Code := 1007;
END_IF;

FOR L_i := 1 TO GVL_CONSTANTS.C_MAX_MANIFOLDS DO
    L_HP_Manifold_Adjusted[L_i] := GVL_CONFIG.G_Manifold_Priority[L_i];
END_FOR;

FOR L_i := 1 TO GVL_CONSTANTS.C_MAX_HEATING_CIRCUITS DO
    L_j := TO_INT(GVL_CONFIG.G_HMI_FloorHeating_Configs[L_i].manifold_id);

    IF (L_j >= 1) AND (L_j <= GVL_CONSTANTS.C_MAX_MANIFOLDS) THEN
        L_HP_Manifold_Adjusted[L_j] := L_HP_Manifold_Adjusted[L_j] + TO_INT(GVL_HEATING_POLICY.G_Zone_Priority_Bias[L_i]);

        IF GVL_HEATING_POLICY_CONFIG.G_Guest_Preheat_Enabled AND GVL_HEATING_POLICY.G_Zone_Guest_Preheat_Request[L_i] THEN
            L_HP_Manifold_Adjusted[L_j] := L_HP_Manifold_Adjusted[L_j] + GVL_HEATING_POLICY_CONFIG.G_Guest_Preheat_Priority_Boost;
        END_IF;

        IF L_HP_Manifold_Adjusted[L_j] < 1 THEN
            GVL_TEST.G_HP_Adjusted_Priority_Lower_Bound_Violation := TRUE;
            GVL_TEST.G_Test_Failed_Checks := GVL_TEST.G_Test_Failed_Checks + 1;
            GVL_TEST.G_Test_Passed := FALSE;
            GVL_TEST.G_Test_Last_Failure_Index := 5;
            GVL_TEST.G_Test_Last_Failure_Code := 1006;
        END_IF;
    END_IF;
END_FOR;

FOR L_i := 1 TO GVL_CONSTANTS.C_MAX_MANIFOLDS DO
    GVL_TEST.G_HP_Manifold_Adjusted_Priority[L_i] := L_HP_Manifold_Adjusted[L_i];
END_FOR;

fbDecisionHP(
    VI_Manifold_Pump_In_Service := GVL_CONFIG.G_Manifold_Pump_In_Service,
    VI_Manifold_Pressure_Fault := GVL_STATUS.G_Diagnostics.Manifold_Pressure_Fault,
    VI_Manifold_Current_Fault := GVL_STATUS.G_Diagnostics.Manifold_Current_Fault,
    VI_Manifold_Thermal_Weight := GVL_CONFIG.G_Manifold_Thermal_Weight,
    VI_Manifold_Priority := L_HP_Manifold_Adjusted,
    VI_Max_Thermal_Budget := GVL_CONFIG.G_Max_Thermal_Budget
);

L_HP_Used := 0.0;
FOR L_i := 1 TO GVL_CONSTANTS.C_MAX_MANIFOLDS DO
    IF fbDecisionHP.VO_Manifold_Enabled[L_i] AND (NOT fbDecisionHP.VO_Manifold_Allowed[L_i]) THEN
        GVL_TEST.G_HP_Adjusted_Allocation_Enabled_Not_Allowed := TRUE;
        GVL_TEST.G_Test_Failed_Checks := GVL_TEST.G_Test_Failed_Checks + 1;
        GVL_TEST.G_Test_Passed := FALSE;
        GVL_TEST.G_Test_Last_Failure_Index := 5;
        GVL_TEST.G_Test_Last_Failure_Code := 1008;
    END_IF;

    IF fbDecisionHP.VO_Manifold_Enabled[L_i] THEN
        L_HP_Used := L_HP_Used + GVL_CONFIG.G_Manifold_Thermal_Weight[L_i];
    END_IF;
END_FOR;

IF L_HP_Used > (GVL_CONFIG.G_Max_Thermal_Budget + 0.001) THEN
    GVL_TEST.G_HP_Adjusted_Allocation_Budget_Exceeded := TRUE;
    GVL_TEST.G_Test_Failed_Checks := GVL_TEST.G_Test_Failed_Checks + 1;
    GVL_TEST.G_Test_Passed := FALSE;
    GVL_TEST.G_Test_Last_Failure_Index := 5;
    GVL_TEST.G_Test_Last_Failure_Code := 1009;
END_IF;

IF GVL_TEST.G_Test_Passed THEN
    GVL_TEST.G_Test_Status_Msg := 'ALL TESTS PASSED';
ELSE
    GVL_TEST.G_Test_Status_Msg := 'TEST FAILURES DETECTED';
END_IF;

fbTestResult(
    VI_Test_Passed := GVL_TEST.G_Test_Passed
);

IF NOT GVL_TEST.G_Test_Passed THEN
    fbTrace(
        VI_Event_Code := UDINT_TO_INT(GVL_TEST.G_Test_Last_Failure_Code),
        VI_System_Time := GVL_STATUS.G_System_Time_MS
    );
END_IF;

(* ---- PRG_Test_Injection.st ---- *)
PROGRAM PRG_Test_Injection

// Non-intrusive test injection layer
// Must be called AFTER PRG_IO_Read and BEFORE PRG_Safety

IF NOT GVL_TEST_INJECTION.G_Inject_Enable THEN
    RETURN;
END_IF;

// ===== GAS INJECTION =====
IF GVL_TEST_INJECTION.G_Inject_Gas_Level > 0.0 THEN
    GVL_STATE.G_Methane_Sensors[1] := GVL_TEST_INJECTION.G_Inject_Gas_Level;
END_IF;

// ===== IO OFFLINE INJECTION =====
IF GVL_TEST_INJECTION.G_Inject_Force_IO_Offline THEN
    GVL_STATUS.G_IO_Modules_Online[1] := FALSE;
    GVL_STATUS.G_IO_Modules_Online[2] := FALSE;
END_IF;

// ===== OWNERSHIP VIOLATION TEST =====
// Intentionally break safety to verify watchdog
IF GVL_TEST_INJECTION.G_Inject_Force_Gas_Alarm_Reset THEN
    GVL_STATE.G_Safety_Gas_Alarm := FALSE;
END_IF;
